KUKA KRL program: f1_Kuka_APT220T03S20.SRC

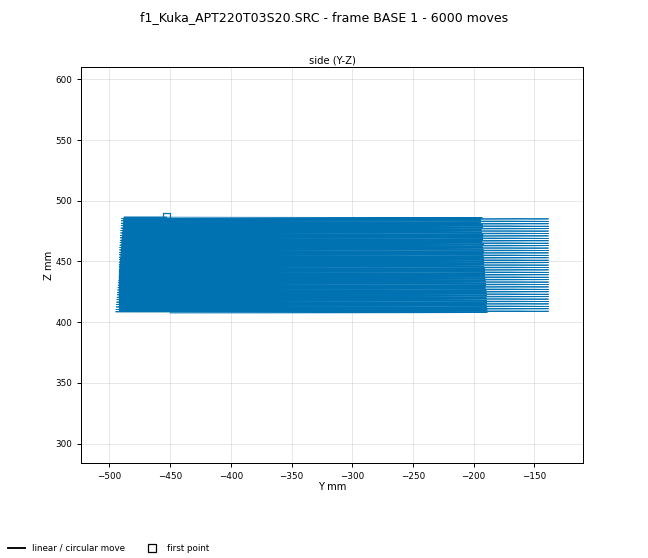
[picture p0: tool path of f1_Kuka_APT220T03S20.SRC in frame BASE 1, 6000 of 6001 moves have a stored position in this frame; points joined in program order, loops and branches not executed]
&ACCESS RVP
&REL 2
&PARAM TEMPLATE = C:\KRC\Roboter\Template\vorgabe
&PARAM EDITMASK = *
DEF f1_Kuka_APT220T03S20()


;FOLD INI;%{PE}%V3.2.0,%MKUKATPBASIS,%CINIT,%VCOMMON,%P
  ;FOLD BAS INI;%{E}%V3.2.0,%MKUKATPBASIS,%CINIT,%VINIT,%P
    GLOBAL INTERRUPT DECL 3 WHEN $STOPMESS==TRUE DO IR_STOPM ( )
    INTERRUPT ON 3
    BAS (#INITMOV,0 )
  ;ENDFOLD (BAS INI)
  ;FOLD USER INI;%{E}%V3.2.0,%MKUKATPUSER,%CINIT,%VINIT,%P
    ;Make your modifications here
  ;ENDFOLD (USER INI)
;ENDFOLD (INI)


;*** Make Null PTP Move
  PTP $pos_act

;*** Auto Load The Correct TOOL Data
  $tool=tool_data[3]

;*** Auto Load The Correct BASE Data
  $base=base_data[1]

  $ADVANCE = 5

;*** Restate Last Velocity
MMPM(30000.0)
SetRPM(6000)
LIN {X -0.066,Y -453.001,Z 486.562,A 0.000,B 0.000,C 90.000,E1 101.130} C_DIS
LIN {X -0.099,Y -473.711,Z 486.551,A 0.000,B 0.000,C 90.000,E1 99.265} C_DIS
LIN {X 0.194,Y -481.469,Z 486.548,A 0.000,B 0.000,C 90.000,E1 98.568} C_DIS
LIN {X 0.203,Y -483.436,Z 486.546,A 0.000,B 0.000,C 90.000,E1 98.341} C_DIS
LIN {X -0.197,Y -484.945,Z 486.545,A 0.000,B 0.000,C 90.000,E1 98.163} C_DIS
LIN {X 0.167,Y -486.209,Z 486.544,A 0.000,B 0.000,C 90.000,E1 97.871} C_DIS
LIN {X -0.015,Y -487.138,Z 486.542,A 0.000,B 0.000,C 90.000,E1 97.644} C_DIS
LIN {X 0.186,Y -488.149,Z 486.540,A 0.000,B 0.000,C 90.000,E1 97.125} C_DIS
LIN {X -0.091,Y -488.162,Z 486.537,A 0.000,B 0.000,C 90.000,E1 96.663} C_DIS
LIN {X 0.122,Y -487.175,Z 486.534,A 0.000,B 0.000,C 90.000,E1 96.144} C_DIS
LIN {X 0.010,Y -486.265,Z 486.533,A 0.000,B 0.000,C 90.000,E1 95.910} C_DIS
LIN {X -0.151,Y -485.019,Z 486.531,A 0.000,B 0.000,C 90.000,E1 95.682} C_DIS
LIN {X 0.212,Y -483.351,Z 486.530,A 0.000,B 0.000,C 90.000,E1 95.391} C_DIS
LIN {X 0.076,Y -465.274,Z 486.518,A 0.000,B 0.000,C 90.000,E1 93.154} C_DIS
LIN {X 0.213,Y -454.119,Z 486.509,A 0.000,B 0.000,C 90.000,E1 91.604} C_DIS
LIN {X 0.144,Y -435.760,Z 486.493,A 0.000,B 0.000,C 90.000,E1 88.740} C_DIS
LIN {X 0.163,Y -421.080,Z 486.480,A 0.000,B 0.000,C 90.000,E1 86.331} C_DIS
LIN {X 0.167,Y -408.275,Z 486.468,A 0.000,B 0.000,C 90.000,E1 84.147} C_DIS
LIN {X -0.037,Y -395.778,Z 486.455,A 0.000,B 0.000,C 90.000,E1 81.951} C_DIS
LIN {X -0.125,Y -384.823,Z 486.444,A 0.000,B 0.000,C 90.000,E1 79.982} C_DIS
LIN {X 0.074,Y -369.281,Z 486.428,A 0.000,B 0.000,C 90.000,E1 77.061} C_DIS
LIN {X 0.055,Y -357.557,Z 486.415,A 0.000,B 0.000,C 90.000,E1 74.700} C_DIS
LIN {X -0.046,Y -347.157,Z 486.402,A 0.000,B 0.000,C 90.000,E1 72.308} C_DIS
LIN {X 0.119,Y -333.448,Z 486.381,A 0.000,B 0.000,C 90.000,E1 68.592} C_DIS
LIN {X 0.012,Y -323.935,Z 486.366,A 0.000,B 0.000,C 90.000,E1 65.793} C_DIS
LIN {X -0.012,Y -315.733,Z 486.351,A 0.000,B 0.000,C 90.000,E1 63.256} C_DIS
LIN {X 0.042,Y -307.567,Z 486.337,A 0.000,B 0.000,C 90.000,E1 60.667} C_DIS
LIN {X 0.124,Y -297.594,Z 486.319,A 0.000,B 0.000,C 90.000,E1 57.375} C_DIS
LIN {X -0.027,Y -288.131,Z 486.300,A 0.000,B 0.000,C 90.000,E1 54.069} C_DIS
LIN {X 0.029,Y -282.669,Z 486.289,A 0.000,B 0.000,C 90.000,E1 52.029} C_DIS
LIN {X -0.014,Y -277.048,Z 486.278,A 0.000,B 0.000,C 90.000,E1 49.989} C_DIS
LIN {X -0.019,Y -270.999,Z 486.266,A 0.000,B 0.000,C 90.000,E1 47.919} C_DIS
LIN {X 0.045,Y -264.538,Z 486.255,A 0.000,B 0.000,C 90.000,E1 45.810} C_DIS
LIN {X -0.028,Y -257.779,Z 486.243,A 0.000,B 0.000,C 90.000,E1 43.704} C_DIS
LIN {X -0.024,Y -248.806,Z 486.227,A 0.000,B 0.000,C 90.000,E1 40.825} C_DIS
LIN {X 0.021,Y -240.234,Z 486.211,A 0.000,B 0.000,C 90.000,E1 37.890} C_DIS
LIN {X 0.095,Y -232.095,Z 486.194,A 0.000,B 0.000,C 90.000,E1 34.898} C_DIS
LIN {X 0.084,Y -224.777,Z 486.177,A 0.000,B 0.000,C 90.000,E1 31.878} C_DIS
LIN {X 0.039,Y -218.459,Z 486.160,A 0.000,B 0.000,C 90.000,E1 28.821} C_DIS
LIN {X 0.011,Y -212.877,Z 486.143,A 0.000,B 0.000,C 90.000,E1 25.720} C_DIS
LIN {X 0.061,Y -207.080,Z 486.121,A 0.000,B 0.000,C 90.000,E1 21.770} C_DIS
LIN {X -0.059,Y -202.295,Z 486.099,A 0.000,B 0.000,C 90.000,E1 17.819} C_DIS
LIN {X 0.019,Y -198.439,Z 486.077,A 0.000,B 0.000,C 90.000,E1 13.772} C_DIS
LIN {X -0.032,Y -195.236,Z 486.049,A 0.000,B 0.000,C 90.000,E1 8.916} C_DIS
LIN {X -0.003,Y -192.924,Z 486.009,A 0.000,B 0.000,C 90.000,E1 1.547} C_DIS
LIN {X 0.083,Y -194.698,Z 485.956,A 0.000,B 0.000,C 90.000,E1 352.129} C_DIS
LIN {X 0.104,Y -197.850,Z 485.929,A 0.000,B 0.000,C 90.000,E1 347.229} C_DIS
LIN {X -0.053,Y -202.300,Z 485.902,A 0.000,B 0.000,C 90.000,E1 342.417} C_DIS
LIN {X -0.067,Y -207.060,Z 485.880,A 0.000,B 0.000,C 90.000,E1 338.411} C_DIS
LIN {X 0.066,Y -212.566,Z 485.858,A 0.000,B 0.000,C 90.000,E1 334.409} C_DIS
LIN {X -0.012,Y -218.738,Z 485.836,A 0.000,B 0.000,C 90.000,E1 330.511} C_DIS
LIN {X 0.052,Y -225.483,Z 485.815,A 0.000,B 0.000,C 90.000,E1 326.628} C_DIS
LIN {X -0.056,Y -232.921,Z 485.793,A 0.000,B 0.000,C 90.000,E1 322.844} C_DIS
LIN {X -0.070,Y -241.150,Z 485.773,A 0.000,B 0.000,C 90.000,E1 319.094} C_DIS
LIN {X -0.057,Y -248.484,Z 485.756,A 0.000,B 0.000,C 90.000,E1 316.134} C_DIS
LIN {X 0.002,Y -257.837,Z 485.738,A 0.000,B 0.000,C 90.000,E1 312.852} C_DIS
LIN {X 0.080,Y -269.299,Z 485.718,A 0.000,B 0.000,C 90.000,E1 309.277} C_DIS
LIN {X 0.060,Y -282.037,Z 485.699,A 0.000,B 0.000,C 90.000,E1 305.804} C_DIS
LIN {X 0.021,Y -295.837,Z 485.680,A 0.000,B 0.000,C 90.000,E1 302.418} C_DIS
LIN {X -0.105,Y -309.070,Z 485.664,A 0.000,B 0.000,C 90.000,E1 299.461} C_DIS
LIN {X -0.041,Y -320.167,Z 485.651,A 0.000,B 0.000,C 90.000,E1 297.180} C_DIS
LIN {X -0.087,Y -336.107,Z 485.635,A 0.000,B 0.000,C 90.000,E1 294.335} C_DIS
LIN {X 0.044,Y -351.864,Z 485.621,A 0.000,B 0.000,C 90.000,E1 291.844} C_DIS
LIN {X -0.013,Y -369.266,Z 485.608,A 0.000,B 0.000,C 90.000,E1 289.450} C_DIS
LIN {X 0.122,Y -388.273,Z 485.595,A 0.000,B 0.000,C 90.000,E1 287.094} C_DIS
LIN {X -0.021,Y -410.726,Z 485.581,A 0.000,B 0.000,C 90.000,E1 284.592} C_DIS
LIN {X -0.224,Y -426.019,Z 485.572,A 0.000,B 0.000,C 90.000,E1 283.008} C_DIS
LIN {X -0.004,Y -438.423,Z 485.565,A 0.000,B 0.000,C 90.000,E1 281.658} C_DIS
LIN {X -0.012,Y -448.140,Z 485.559,A 0.000,B 0.000,C 90.000,E1 280.602} C_DIS
LIN {X 0.192,Y -454.892,Z 485.555,A 0.000,B 0.000,C 90.000,E1 279.792} C_DIS
LIN {X 0.079,Y -461.053,Z 485.550,A 0.000,B 0.000,C 90.000,E1 279.029} C_DIS
LIN {X -0.054,Y -466.674,Z 485.546,A 0.000,B 0.000,C 90.000,E1 278.276} C_DIS
LIN {X -0.208,Y -471.720,Z 485.542,A 0.000,B 0.000,C 90.000,E1 277.530} C_DIS
LIN {X 0.223,Y -476.192,Z 485.537,A 0.000,B 0.000,C 90.000,E1 276.720} C_DIS
LIN {X 0.215,Y -480.149,Z 485.533,A 0.000,B 0.000,C 90.000,E1 275.967} C_DIS
LIN {X -0.156,Y -482.500,Z 485.531,A 0.000,B 0.000,C 90.000,E1 275.511} C_DIS
LIN {X 0.016,Y -484.512,Z 485.528,A 0.000,B 0.000,C 90.000,E1 274.992} C_DIS
LIN {X 0.193,Y -486.239,Z 485.525,A 0.000,B 0.000,C 90.000,E1 274.473} C_DIS
LIN {X -0.105,Y -487.676,Z 485.522,A 0.000,B 0.000,C 90.000,E1 274.012} C_DIS
LIN {X 0.058,Y -488.770,Z 485.519,A 0.000,B 0.000,C 90.000,E1 273.498} C_DIS
LIN {X -0.227,Y -489.533,Z 485.517,A 0.000,B 0.000,C 90.000,E1 273.037} C_DIS
LIN {X -0.044,Y -489.993,Z 485.514,A 0.000,B 0.000,C 90.000,E1 272.522} C_DIS
LIN {X 0.146,Y -490.072,Z 485.511,A 0.000,B 0.000,C 90.000,E1 272.007} C_DIS
LIN {X -0.134,Y -489.708,Z 485.509,A 0.000,B 0.000,C 90.000,E1 271.547} C_DIS
LIN {X 0.060,Y -488.939,Z 485.506,A 0.000,B 0.000,C 90.000,E1 271.031} C_DIS
LIN {X -0.235,Y -487.615,Z 485.503,A 0.000,B 0.000,C 90.000,E1 270.573} C_DIS
LIN {X -0.046,Y -485.714,Z 485.500,A 0.000,B 0.000,C 90.000,E1 270.057} C_DIS
LIN {X 0.134,Y -483.153,Z 485.498,A 0.000,B 0.000,C 90.000,E1 269.542} C_DIS
LIN {X -0.186,Y -479.844,Z 485.495,A 0.000,B 0.000,C 90.000,E1 269.083} C_DIS
LIN {X -0.043,Y -475.615,Z 485.492,A 0.000,B 0.000,C 90.000,E1 268.568} C_DIS
LIN {X 0.091,Y -470.396,Z 485.489,A 0.000,B 0.000,C 90.000,E1 268.051} C_DIS
LIN {X 0.002,Y -464.305,Z 485.487,A 0.000,B 0.000,C 90.000,E1 267.593} C_DIS
LIN {X -0.231,Y -461.262,Z 485.486,A 0.000,B 0.000,C 90.000,E1 267.421} C_DIS
LIN {X 0.033,Y -454.595,Z 485.483,A 0.000,B 0.000,C 90.000,E1 267.020} C_DIS
LIN {X -0.113,Y -447.751,Z 485.482,A 0.000,B 0.000,C 90.000,E1 266.731} C_DIS
LIN {X 0.088,Y -440.644,Z 485.480,A 0.000,B 0.000,C 90.000,E1 266.445} C_DIS
LIN {X -0.218,Y -432.837,Z 485.479,A 0.000,B 0.000,C 90.000,E1 266.274} C_DIS
LIN {X -0.101,Y -424.190,Z 485.478,A 0.000,B 0.000,C 90.000,E1 266.102} C_DIS
LIN {X -0.056,Y -413.858,Z 485.478,A 0.000,B 0.000,C 90.000,E1 265.988} C_DIS
LIN {X -0.214,Y -409.409,Z 485.478,A 0.000,B 0.000,C 90.000,E1 265.988} C_DIS
LIN {X 0.063,Y -180.918,Z 485.477,A 0.000,B 0.000,C 90.000,E1 265.927} C_DIS
LIN {X -0.088,Y -180.843,Z 485.472,A 0.000,B 0.000,C 90.000,E1 264.951} C_DIS
LIN {X -0.011,Y -178.885,Z 485.443,A 0.000,B 0.000,C 90.000,E1 259.690} C_DIS
LIN {X 0.064,Y -175.928,Z 485.414,A 0.000,B 0.000,C 90.000,E1 254.574} C_DIS
LIN {X 0.009,Y -175.370,Z 485.410,A 0.000,B 0.000,C 90.000,E1 253.740} C_DIS
LIN {X 0.067,Y -172.147,Z 485.386,A 0.000,B 0.000,C 90.000,E1 249.444} C_DIS
LIN {X 0.045,Y -171.612,Z 485.381,A 0.000,B 0.000,C 90.000,E1 248.592} C_DIS
LIN {X 0.033,Y -167.834,Z 485.357,A 0.000,B 0.000,C 90.000,E1 244.280} C_DIS
LIN {X 0.050,Y -166.561,Z 485.348,A 0.000,B 0.000,C 90.000,E1 242.538} C_DIS
LIN {X -0.040,Y -162.555,Z 485.323,A 0.000,B 0.000,C 90.000,E1 238.201} C_DIS
LIN {X 0.020,Y -161.234,Z 485.313,A 0.000,B 0.000,C 90.000,E1 236.421} C_DIS
LIN {X 0.054,Y -157.239,Z 485.289,A 0.000,B 0.000,C 90.000,E1 231.984} C_DIS
LIN {X -0.022,Y -155.962,Z 485.279,A 0.000,B 0.000,C 90.000,E1 230.231} C_DIS
LIN {X 0.036,Y -152.217,Z 485.254,A 0.000,B 0.000,C 90.000,E1 225.729} C_DIS
LIN {X 0.056,Y -150.461,Z 485.239,A 0.000,B 0.000,C 90.000,E1 223.014} C_DIS
LIN {X 0.082,Y -147.186,Z 485.214,A 0.000,B 0.000,C 90.000,E1 218.463} C_DIS
LIN {X 0.049,Y -145.204,Z 485.194,A 0.000,B 0.000,C 90.000,E1 214.818} C_DIS
LIN {X -0.041,Y -142.340,Z 485.163,A 0.000,B 0.000,C 90.000,E1 209.333} C_DIS
LIN {X 0.012,Y -141.728,Z 485.153,A 0.000,B 0.000,C 90.000,E1 207.462} C_DIS
LIN {X -0.006,Y -139.482,Z 485.116,A 0.000,B 0.000,C 90.000,E1 200.972} C_DIS
LIN {X -0.017,Y -138.980,Z 485.101,A 0.000,B 0.000,C 90.000,E1 198.181} C_DIS
LIN {X -0.056,Y -138.333,Z 485.054,A 0.000,B 0.000,C 90.000,E1 189.792} C_DIS
LIN {X -0.032,Y -139.428,Z 485.008,A 0.000,B 0.000,C 90.000,E1 181.375} C_DIS
LIN {X 0.022,Y -141.355,Z 484.971,A 0.000,B 0.000,C 90.000,E1 174.837} C_DIS
LIN {X -0.002,Y -142.708,Z 484.956,A 0.000,B 0.000,C 90.000,E1 172.064} C_DIS
LIN {X -0.043,Y -145.082,Z 484.930,A 0.000,B 0.000,C 90.000,E1 167.465} C_DIS
LIN {X -0.047,Y -147.707,Z 484.910,A 0.000,B 0.000,C 90.000,E1 163.795} C_DIS
LIN {X 0.036,Y -150.361,Z 484.890,A 0.000,B 0.000,C 90.000,E1 160.115} C_DIS
LIN {X 0.054,Y -153.786,Z 484.869,A 0.000,B 0.000,C 90.000,E1 156.485} C_DIS
LIN {X -0.025,Y -157.198,Z 484.850,A 0.000,B 0.000,C 90.000,E1 152.922} C_DIS
LIN {X 0.057,Y -161.360,Z 484.830,A 0.000,B 0.000,C 90.000,E1 149.331} C_DIS
LIN {X 0.068,Y -165.562,Z 484.810,A 0.000,B 0.000,C 90.000,E1 145.801} C_DIS
LIN {X -0.048,Y -170.478,Z 484.791,A 0.000,B 0.000,C 90.000,E1 142.351} C_DIS
LIN {X 0.101,Y -175.360,Z 484.772,A 0.000,B 0.000,C 90.000,E1 138.852} C_DIS
LIN {X -0.035,Y -180.985,Z 484.753,A 0.000,B 0.000,C 90.000,E1 135.486} C_DIS
LIN {X -0.049,Y -186.409,Z 484.734,A 0.000,B 0.000,C 90.000,E1 132.123} C_DIS
LIN {X -0.110,Y -191.038,Z 484.720,A 0.000,B 0.000,C 90.000,E1 129.644} C_DIS
LIN {X 0.023,Y -193.423,Z 484.712,A 0.000,B 0.000,C 90.000,E1 128.177} C_DIS
LIN {X -0.005,Y -291.168,Z 484.712,A 0.000,B 0.000,C 90.000,E1 128.177} C_DIS
LIN {X -0.085,Y -292.124,Z 484.712,A 0.000,B 0.000,C 90.000,E1 128.177} C_DIS
LIN {X -0.050,Y -296.671,Z 484.711,A 0.000,B 0.000,C 90.000,E1 127.971} C_DIS
LIN {X 0.020,Y -299.838,Z 484.709,A 0.000,B 0.000,C 90.000,E1 127.684} C_DIS
LIN {X 0.147,Y -303.532,Z 484.707,A 0.000,B 0.000,C 90.000,E1 127.156} C_DIS
LIN {X -0.090,Y -305.238,Z 484.705,A 0.000,B 0.000,C 90.000,E1 126.870} C_DIS
LIN {X 0.101,Y -306.580,Z 484.703,A 0.000,B 0.000,C 90.000,E1 126.503} C_DIS
LIN {X -0.077,Y -317.797,Z 484.683,A 0.000,B 0.000,C 90.000,E1 122.959} C_DIS
LIN {X -0.030,Y -328.281,Z 484.667,A 0.000,B 0.000,C 90.000,E1 120.079} C_DIS
LIN {X -0.002,Y -340.128,Z 484.651,A 0.000,B 0.000,C 90.000,E1 117.257} C_DIS
LIN {X -0.116,Y -353.449,Z 484.636,A 0.000,B 0.000,C 90.000,E1 114.515} C_DIS
LIN {X 0.108,Y -366.623,Z 484.623,A 0.000,B 0.000,C 90.000,E1 112.078} C_DIS
LIN {X -0.082,Y -381.150,Z 484.610,A 0.000,B 0.000,C 90.000,E1 109.758} C_DIS
LIN {X -0.040,Y -397.136,Z 484.597,A 0.000,B 0.000,C 90.000,E1 107.457} C_DIS
LIN {X 0.171,Y -414.700,Z 484.585,A 0.000,B 0.000,C 90.000,E1 105.190} C_DIS
LIN {X -0.185,Y -433.943,Z 484.572,A 0.000,B 0.000,C 90.000,E1 103.063} C_DIS
LIN {X 0.027,Y -454.145,Z 484.561,A 0.000,B 0.000,C 90.000,E1 101.007} C_DIS
LIN {X -0.012,Y -474.885,Z 484.551,A 0.000,B 0.000,C 90.000,E1 99.151} C_DIS
LIN {X 0.167,Y -480.145,Z 484.548,A 0.000,B 0.000,C 90.000,E1 98.690} C_DIS
LIN {X -0.145,Y -482.402,Z 484.547,A 0.000,B 0.000,C 90.000,E1 98.511} C_DIS
LIN {X 0.018,Y -484.116,Z 484.546,A 0.000,B 0.000,C 90.000,E1 98.276} C_DIS
LIN {X -0.170,Y -485.628,Z 484.545,A 0.000,B 0.000,C 90.000,E1 98.049} C_DIS
LIN {X 0.193,Y -486.758,Z 484.543,A 0.000,B 0.000,C 90.000,E1 97.757} C_DIS
LIN {X -0.095,Y -488.102,Z 484.540,A 0.000,B 0.000,C 90.000,E1 97.296} C_DIS
LIN {X 0.109,Y -488.413,Z 484.538,A 0.000,B 0.000,C 90.000,E1 96.777} C_DIS
LIN {X -0.164,Y -487.742,Z 484.535,A 0.000,B 0.000,C 90.000,E1 96.315} C_DIS
LIN {X 0.049,Y -485.978,Z 484.532,A 0.000,B 0.000,C 90.000,E1 95.796} C_DIS
LIN {X -0.112,Y -484.583,Z 484.531,A 0.000,B 0.000,C 90.000,E1 95.568} C_DIS
LIN {X -0.079,Y -478.706,Z 484.527,A 0.000,B 0.000,C 90.000,E1 94.821} C_DIS
LIN {X 0.175,Y -460.878,Z 484.514,A 0.000,B 0.000,C 90.000,E1 92.522} C_DIS
LIN {X -0.020,Y -448.423,Z 484.504,A 0.000,B 0.000,C 90.000,E1 90.745} C_DIS
LIN {X 0.149,Y -435.261,Z 484.492,A 0.000,B 0.000,C 90.000,E1 88.625} C_DIS
LIN {X 0.149,Y -420.581,Z 484.479,A 0.000,B 0.000,C 90.000,E1 86.216} C_DIS
LIN {X -0.158,Y -406.238,Z 484.465,A 0.000,B 0.000,C 90.000,E1 83.799} C_DIS
LIN {X -0.078,Y -395.315,Z 484.455,A 0.000,B 0.000,C 90.000,E1 81.837} C_DIS
LIN {X -0.108,Y -384.376,Z 484.444,A 0.000,B 0.000,C 90.000,E1 79.859} C_DIS
LIN {X 0.088,Y -368.860,Z 484.427,A 0.000,B 0.000,C 90.000,E1 76.937} C_DIS
LIN {X 0.066,Y -357.181,Z 484.414,A 0.000,B 0.000,C 90.000,E1 74.574} C_DIS
LIN {X -0.038,Y -346.833,Z 484.401,A 0.000,B 0.000,C 90.000,E1 72.181} C_DIS
LIN {X 0.131,Y -334.216,Z 484.382,A 0.000,B 0.000,C 90.000,E1 68.773} C_DIS
LIN {X -0.036,Y -322.537,Z 484.363,A 0.000,B 0.000,C 90.000,E1 65.357} C_DIS
LIN {X 0.044,Y -316.364,Z 484.352,A 0.000,B 0.000,C 90.000,E1 63.435} C_DIS
LIN {X 0.118,Y -308.153,Z 484.338,A 0.000,B 0.000,C 90.000,E1 60.845} C_DIS
LIN {X 0.068,Y -298.121,Z 484.320,A 0.000,B 0.000,C 90.000,E1 57.582} C_DIS
LIN {X -0.065,Y -288.589,Z 484.301,A 0.000,B 0.000,C 90.000,E1 54.276} C_DIS
LIN {X -0.172,Y -283.117,Z 484.290,A 0.000,B 0.000,C 90.000,E1 52.271} C_DIS
LIN {X -0.029,Y -277.516,Z 484.279,A 0.000,B 0.000,C 90.000,E1 50.194} C_DIS
LIN {X 0.000,Y -271.503,Z 484.267,A 0.000,B 0.000,C 90.000,E1 48.119} C_DIS
LIN {X -0.126,Y -265.082,Z 484.256,A 0.000,B 0.000,C 90.000,E1 46.053} C_DIS
LIN {X 0.003,Y -258.374,Z 484.244,A 0.000,B 0.000,C 90.000,E1 43.905} C_DIS
LIN {X 0.018,Y -248.304,Z 484.226,A 0.000,B 0.000,C 90.000,E1 40.663} C_DIS
LIN {X 0.027,Y -238.693,Z 484.208,A 0.000,B 0.000,C 90.000,E1 37.363} C_DIS
LIN {X -0.075,Y -230.694,Z 484.191,A 0.000,B 0.000,C 90.000,E1 34.405} C_DIS
LIN {X 0.071,Y -223.578,Z 484.174,A 0.000,B 0.000,C 90.000,E1 31.337} C_DIS
LIN {X -0.007,Y -217.384,Z 484.157,A 0.000,B 0.000,C 90.000,E1 28.281} C_DIS
LIN {X 0.032,Y -211.971,Z 484.140,A 0.000,B 0.000,C 90.000,E1 25.155} C_DIS
LIN {X -0.023,Y -206.290,Z 484.118,A 0.000,B 0.000,C 90.000,E1 21.227} C_DIS
LIN {X 0.032,Y -201.634,Z 484.096,A 0.000,B 0.000,C 90.000,E1 17.221} C_DIS
LIN {X 0.086,Y -197.927,Z 484.073,A 0.000,B 0.000,C 90.000,E1 13.175} C_DIS
LIN {X -0.077,Y -194.481,Z 484.042,A 0.000,B 0.000,C 90.000,E1 7.530} C_DIS
LIN {X 0.057,Y -195.445,Z 483.947,A 0.000,B 0.000,C 90.000,E1 350.500} C_DIS
LIN {X -0.044,Y -199.071,Z 483.920,A 0.000,B 0.000,C 90.000,E1 345.644} C_DIS
LIN {X 0.033,Y -203.010,Z 483.898,A 0.000,B 0.000,C 90.000,E1 341.583} C_DIS
LIN {X -0.007,Y -207.968,Z 483.875,A 0.000,B 0.000,C 90.000,E1 337.592} C_DIS
LIN {X -0.031,Y -213.585,Z 483.854,A 0.000,B 0.000,C 90.000,E1 333.640} C_DIS
LIN {X -0.084,Y -219.884,Z 483.832,A 0.000,B 0.000,C 90.000,E1 329.744} C_DIS
LIN {X -0.064,Y -226.774,Z 483.810,A 0.000,B 0.000,C 90.000,E1 325.881} C_DIS
LIN {X -0.005,Y -234.402,Z 483.789,A 0.000,B 0.000,C 90.000,E1 322.065} C_DIS
LIN {X -0.003,Y -242.796,Z 483.768,A 0.000,B 0.000,C 90.000,E1 318.324} C_DIS
LIN {X 0.052,Y -251.380,Z 483.750,A 0.000,B 0.000,C 90.000,E1 315.000} C_DIS
LIN {X 0.027,Y -261.066,Z 483.732,A 0.000,B 0.000,C 90.000,E1 311.757} C_DIS
LIN {X -0.046,Y -271.684,Z 483.714,A 0.000,B 0.000,C 90.000,E1 308.588} C_DIS
LIN {X 0.061,Y -284.676,Z 483.695,A 0.000,B 0.000,C 90.000,E1 305.105} C_DIS
LIN {X -0.053,Y -298.724,Z 483.676,A 0.000,B 0.000,C 90.000,E1 301.750} C_DIS
LIN {X 0.073,Y -313.690,Z 483.658,A 0.000,B 0.000,C 90.000,E1 298.437} C_DIS
LIN {X 0.169,Y -323.588,Z 483.647,A 0.000,B 0.000,C 90.000,E1 296.488} C_DIS
LIN {X -0.070,Y -339.930,Z 483.632,A 0.000,B 0.000,C 90.000,E1 293.695} C_DIS
LIN {X -0.008,Y -353.980,Z 483.620,A 0.000,B 0.000,C 90.000,E1 291.535} C_DIS
LIN {X -0.099,Y -369.308,Z 483.608,A 0.000,B 0.000,C 90.000,E1 289.450} C_DIS
LIN {X 0.033,Y -388.293,Z 483.595,A 0.000,B 0.000,C 90.000,E1 287.094} C_DIS
LIN {X -0.109,Y -410.777,Z 483.581,A 0.000,B 0.000,C 90.000,E1 284.592} C_DIS
LIN {X -0.177,Y -425.949,Z 483.572,A 0.000,B 0.000,C 90.000,E1 283.008} C_DIS
LIN {X 0.129,Y -438.298,Z 483.565,A 0.000,B 0.000,C 90.000,E1 281.658} C_DIS
LIN {X -0.049,Y -445.608,Z 483.560,A 0.000,B 0.000,C 90.000,E1 280.894} C_DIS
LIN {X 0.157,Y -452.543,Z 483.556,A 0.000,B 0.000,C 90.000,E1 280.084} C_DIS
LIN {X 0.032,Y -458.939,Z 483.552,A 0.000,B 0.000,C 90.000,E1 279.321} C_DIS
LIN {X 0.168,Y -466.548,Z 483.546,A 0.000,B 0.000,C 90.000,E1 278.276} C_DIS
LIN {X 0.015,Y -471.623,Z 483.542,A 0.000,B 0.000,C 90.000,E1 277.530} C_DIS
LIN {X -0.026,Y -476.156,Z 483.538,A 0.000,B 0.000,C 90.000,E1 276.777} C_DIS
LIN {X -0.088,Y -480.145,Z 483.533,A 0.000,B 0.000,C 90.000,E1 276.030} C_DIS
LIN {X 0.070,Y -482.488,Z 483.531,A 0.000,B 0.000,C 90.000,E1 275.511} C_DIS
LIN {X -0.241,Y -484.529,Z 483.528,A 0.000,B 0.000,C 90.000,E1 275.049} C_DIS
LIN {X -0.064,Y -486.287,Z 483.525,A 0.000,B 0.000,C 90.000,E1 274.531} C_DIS
LIN {X 0.123,Y -487.727,Z 483.522,A 0.000,B 0.000,C 90.000,E1 274.012} C_DIS
LIN {X -0.201,Y -488.884,Z 483.520,A 0.000,B 0.000,C 90.000,E1 273.555} C_DIS
LIN {X 0.002,Y -489.645,Z 483.517,A 0.000,B 0.000,C 90.000,E1 273.037} C_DIS
LIN {X 0.186,Y -490.105,Z 483.514,A 0.000,B 0.000,C 90.000,E1 272.522} C_DIS
LIN {X -0.113,Y -490.201,Z 483.511,A 0.000,B 0.000,C 90.000,E1 272.064} C_DIS
LIN {X 0.098,Y -489.875,Z 483.509,A 0.000,B 0.000,C 90.000,E1 271.547} C_DIS
LIN {X -0.197,Y -489.145,Z 483.506,A 0.000,B 0.000,C 90.000,E1 271.088} C_DIS
LIN {X -0.003,Y -487.837,Z 483.503,A 0.000,B 0.000,C 90.000,E1 270.573} C_DIS
LIN {X 0.187,Y -485.979,Z 483.500,A 0.000,B 0.000,C 90.000,E1 270.057} C_DIS
LIN {X -0.116,Y -483.442,Z 483.498,A 0.000,B 0.000,C 90.000,E1 269.599} C_DIS
LIN {X 0.047,Y -480.160,Z 483.495,A 0.000,B 0.000,C 90.000,E1 269.083} C_DIS
LIN {X -0.120,Y -478.231,Z 483.494,A 0.000,B 0.000,C 90.000,E1 268.854} C_DIS
LIN {X 0.013,Y -473.551,Z 483.491,A 0.000,B 0.000,C 90.000,E1 268.339} C_DIS
LIN {X -0.187,Y -468.011,Z 483.488,A 0.000,B 0.000,C 90.000,E1 267.879} C_DIS
LIN {X -0.007,Y -461.773,Z 483.486,A 0.000,B 0.000,C 90.000,E1 267.421} C_DIS
LIN {X 0.218,Y -455.153,Z 483.484,A 0.000,B 0.000,C 90.000,E1 267.020} C_DIS
LIN {X 0.020,Y -448.307,Z 483.482,A 0.000,B 0.000,C 90.000,E1 266.731} C_DIS
LIN {X 0.175,Y -441.166,Z 483.480,A 0.000,B 0.000,C 90.000,E1 266.445} C_DIS
LIN {X -0.151,Y -433.386,Z 483.479,A 0.000,B 0.000,C 90.000,E1 266.274} C_DIS
LIN {X -0.038,Y -425.010,Z 483.478,A 0.000,B 0.000,C 90.000,E1 266.102} C_DIS
LIN {X 0.004,Y -415.303,Z 483.478,A 0.000,B 0.000,C 90.000,E1 265.988} C_DIS
LIN {X 0.175,Y -409.435,Z 483.478,A 0.000,B 0.000,C 90.000,E1 265.931} C_DIS
LIN {X 0.055,Y -180.918,Z 483.477,A 0.000,B 0.000,C 90.000,E1 265.927} C_DIS
LIN {X 0.085,Y -180.842,Z 483.472,A 0.000,B 0.000,C 90.000,E1 264.894} C_DIS
LIN {X -0.019,Y -178.885,Z 483.443,A 0.000,B 0.000,C 90.000,E1 259.690} C_DIS
LIN {X 0.058,Y -175.927,Z 483.414,A 0.000,B 0.000,C 90.000,E1 254.574} C_DIS
LIN {X 0.003,Y -175.368,Z 483.410,A 0.000,B 0.000,C 90.000,E1 253.740} C_DIS
LIN {X 0.061,Y -172.145,Z 483.386,A 0.000,B 0.000,C 90.000,E1 249.444} C_DIS
LIN {X 0.039,Y -171.610,Z 483.381,A 0.000,B 0.000,C 90.000,E1 248.592} C_DIS
LIN {X 0.026,Y -167.833,Z 483.357,A 0.000,B 0.000,C 90.000,E1 244.280} C_DIS
LIN {X 0.044,Y -166.559,Z 483.348,A 0.000,B 0.000,C 90.000,E1 242.538} C_DIS
LIN {X -0.046,Y -162.553,Z 483.323,A 0.000,B 0.000,C 90.000,E1 238.201} C_DIS
LIN {X 0.014,Y -161.232,Z 483.313,A 0.000,B 0.000,C 90.000,E1 236.421} C_DIS
LIN {X 0.049,Y -157.237,Z 483.289,A 0.000,B 0.000,C 90.000,E1 231.984} C_DIS
LIN {X -0.028,Y -155.962,Z 483.279,A 0.000,B 0.000,C 90.000,E1 230.231} C_DIS
LIN {X 0.030,Y -152.215,Z 483.254,A 0.000,B 0.000,C 90.000,E1 225.729} C_DIS
LIN {X 0.051,Y -150.460,Z 483.239,A 0.000,B 0.000,C 90.000,E1 223.014} C_DIS
LIN {X 0.077,Y -147.184,Z 483.214,A 0.000,B 0.000,C 90.000,E1 218.463} C_DIS
LIN {X 0.043,Y -145.203,Z 483.194,A 0.000,B 0.000,C 90.000,E1 214.818} C_DIS
LIN {X -0.047,Y -142.339,Z 483.163,A 0.000,B 0.000,C 90.000,E1 209.333} C_DIS
LIN {X 0.006,Y -141.727,Z 483.153,A 0.000,B 0.000,C 90.000,E1 207.462} C_DIS
LIN {X -0.012,Y -139.480,Z 483.116,A 0.000,B 0.000,C 90.000,E1 200.972} C_DIS
LIN {X -0.022,Y -138.980,Z 483.101,A 0.000,B 0.000,C 90.000,E1 198.181} C_DIS
LIN {X -0.038,Y -138.332,Z 483.054,A 0.000,B 0.000,C 90.000,E1 189.782} C_DIS
LIN {X -0.037,Y -139.428,Z 483.008,A 0.000,B 0.000,C 90.000,E1 181.375} C_DIS
LIN {X 0.016,Y -141.355,Z 482.971,A 0.000,B 0.000,C 90.000,E1 174.837} C_DIS
LIN {X -0.008,Y -142.709,Z 482.956,A 0.000,B 0.000,C 90.000,E1 172.064} C_DIS
LIN {X -0.049,Y -145.083,Z 482.930,A 0.000,B 0.000,C 90.000,E1 167.465} C_DIS
LIN {X -0.053,Y -147.708,Z 482.910,A 0.000,B 0.000,C 90.000,E1 163.795} C_DIS
LIN {X 0.031,Y -150.363,Z 482.890,A 0.000,B 0.000,C 90.000,E1 160.115} C_DIS
LIN {X 0.049,Y -153.788,Z 482.869,A 0.000,B 0.000,C 90.000,E1 156.485} C_DIS
LIN {X -0.031,Y -157.201,Z 482.850,A 0.000,B 0.000,C 90.000,E1 152.922} C_DIS
LIN {X 0.050,Y -161.362,Z 482.830,A 0.000,B 0.000,C 90.000,E1 149.331} C_DIS
LIN {X 0.062,Y -165.565,Z 482.810,A 0.000,B 0.000,C 90.000,E1 145.801} C_DIS
LIN {X -0.054,Y -170.482,Z 482.791,A 0.000,B 0.000,C 90.000,E1 142.351} C_DIS
LIN {X 0.095,Y -175.363,Z 482.772,A 0.000,B 0.000,C 90.000,E1 138.852} C_DIS
LIN {X -0.042,Y -180.987,Z 482.753,A 0.000,B 0.000,C 90.000,E1 135.486} C_DIS
LIN {X -0.055,Y -186.413,Z 482.734,A 0.000,B 0.000,C 90.000,E1 132.123} C_DIS
LIN {X -0.116,Y -191.041,Z 482.720,A 0.000,B 0.000,C 90.000,E1 129.644} C_DIS
LIN {X -0.116,Y -193.495,Z 482.712,A 0.000,B 0.000,C 90.000,E1 128.177} C_DIS
LIN {X -0.030,Y -290.585,Z 482.712,A 0.000,B 0.000,C 90.000,E1 128.141} C_DIS
LIN {X -0.060,Y -296.092,Z 482.711,A 0.000,B 0.000,C 90.000,E1 127.971} C_DIS
LIN {X 0.019,Y -299.041,Z 482.710,A 0.000,B 0.000,C 90.000,E1 127.729} C_DIS
LIN {X -0.027,Y -302.787,Z 482.707,A 0.000,B 0.000,C 90.000,E1 127.282} C_DIS
LIN {X -0.005,Y -304.668,Z 482.705,A 0.000,B 0.000,C 90.000,E1 126.950} C_DIS
LIN {X -0.044,Y -306.141,Z 482.703,A 0.000,B 0.000,C 90.000,E1 126.629} C_DIS
LIN {X 0.005,Y -308.271,Z 482.700,A 0.000,B 0.000,C 90.000,E1 125.964} C_DIS
LIN {X -0.181,Y -318.545,Z 482.682,A 0.000,B 0.000,C 90.000,E1 122.752} C_DIS
LIN {X -0.113,Y -329.129,Z 482.666,A 0.000,B 0.000,C 90.000,E1 119.873} C_DIS
LIN {X -0.073,Y -341.089,Z 482.650,A 0.000,B 0.000,C 90.000,E1 117.052} C_DIS
LIN {X 0.157,Y -354.525,Z 482.635,A 0.000,B 0.000,C 90.000,E1 114.259} C_DIS
LIN {X -0.062,Y -367.813,Z 482.622,A 0.000,B 0.000,C 90.000,E1 111.897} C_DIS
LIN {X -0.227,Y -382.462,Z 482.609,A 0.000,B 0.000,C 90.000,E1 109.577} C_DIS
LIN {X -0.157,Y -398.581,Z 482.596,A 0.000,B 0.000,C 90.000,E1 107.275} C_DIS
LIN {X 0.085,Y -416.289,Z 482.583,A 0.000,B 0.000,C 90.000,E1 105.009} C_DIS
LIN {X 0.211,Y -435.653,Z 482.571,A 0.000,B 0.000,C 90.000,E1 102.827} C_DIS
LIN {X 0.027,Y -455.904,Z 482.560,A 0.000,B 0.000,C 90.000,E1 100.838} C_DIS
LIN {X 0.187,Y -476.687,Z 482.550,A 0.000,B 0.000,C 90.000,E1 98.973} C_DIS
LIN {X -0.083,Y -481.803,Z 482.548,A 0.000,B 0.000,C 90.000,E1 98.568} C_DIS
LIN {X 0.003,Y -483.695,Z 482.546,A 0.000,B 0.000,C 90.000,E1 98.341} C_DIS
LIN {X -0.115,Y -485.352,Z 482.545,A 0.000,B 0.000,C 90.000,E1 98.106} C_DIS
LIN {X 0.246,Y -486.593,Z 482.544,A 0.000,B 0.000,C 90.000,E1 97.814} C_DIS
LIN {X -0.044,Y -488.115,Z 482.541,A 0.000,B 0.000,C 90.000,E1 97.352} C_DIS
LIN {X 0.158,Y -488.580,Z 482.538,A 0.000,B 0.000,C 90.000,E1 96.834} C_DIS
LIN {X -0.116,Y -488.067,Z 482.535,A 0.000,B 0.000,C 90.000,E1 96.372} C_DIS
LIN {X 0.098,Y -486.491,Z 482.533,A 0.000,B 0.000,C 90.000,E1 95.853} C_DIS
LIN {X -0.064,Y -485.218,Z 482.531,A 0.000,B 0.000,C 90.000,E1 95.625} C_DIS
LIN {X -0.176,Y -483.519,Z 482.530,A 0.000,B 0.000,C 90.000,E1 95.391} C_DIS
LIN {X -0.188,Y -471.414,Z 482.522,A 0.000,B 0.000,C 90.000,E1 93.898} C_DIS
LIN {X 0.063,Y -456.086,Z 482.510,A 0.000,B 0.000,C 90.000,E1 91.835} C_DIS
LIN {X -0.027,Y -442.447,Z 482.499,A 0.000,B 0.000,C 90.000,E1 89.771} C_DIS
LIN {X -0.136,Y -430.960,Z 482.488,A 0.000,B 0.000,C 90.000,E1 87.936} C_DIS
LIN {X 0.190,Y -416.384,Z 482.475,A 0.000,B 0.000,C 90.000,E1 85.469} C_DIS
LIN {X 0.167,Y -402.173,Z 482.461,A 0.000,B 0.000,C 90.000,E1 82.996} C_DIS
LIN {X -0.180,Y -391.229,Z 482.450,A 0.000,B 0.000,C 90.000,E1 81.084} C_DIS
LIN {X 0.049,Y -381.864,Z 482.441,A 0.000,B 0.000,C 90.000,E1 79.342} C_DIS
LIN {X -0.124,Y -366.477,Z 482.425,A 0.000,B 0.000,C 90.000,E1 76.464} C_DIS
LIN {X -0.149,Y -356.400,Z 482.413,A 0.000,B 0.000,C 90.000,E1 74.393} C_DIS
LIN {X 0.066,Y -346.149,Z 482.400,A 0.000,B 0.000,C 90.000,E1 71.945} C_DIS
LIN {X -0.097,Y -334.674,Z 482.383,A 0.000,B 0.000,C 90.000,E1 68.901} C_DIS
LIN {X 0.043,Y -322.904,Z 482.364,A 0.000,B 0.000,C 90.000,E1 65.433} C_DIS
LIN {X 0.124,Y -314.607,Z 482.349,A 0.000,B 0.000,C 90.000,E1 62.871} C_DIS
LIN {X -0.124,Y -306.373,Z 482.335,A 0.000,B 0.000,C 90.000,E1 60.333} C_DIS
LIN {X 0.145,Y -298.342,Z 482.320,A 0.000,B 0.000,C 90.000,E1 57.661} C_DIS
LIN {X 0.012,Y -288.765,Z 482.302,A 0.000,B 0.000,C 90.000,E1 54.356} C_DIS
LIN {X -0.095,Y -283.285,Z 482.291,A 0.000,B 0.000,C 90.000,E1 52.351} C_DIS
LIN {X 0.048,Y -277.686,Z 482.279,A 0.000,B 0.000,C 90.000,E1 50.275} C_DIS
LIN {X -0.126,Y -271.678,Z 482.268,A 0.000,B 0.000,C 90.000,E1 48.243} C_DIS
LIN {X -0.049,Y -265.292,Z 482.256,A 0.000,B 0.000,C 90.000,E1 46.134} C_DIS
LIN {X -0.104,Y -258.606,Z 482.244,A 0.000,B 0.000,C 90.000,E1 44.028} C_DIS
LIN {X -0.059,Y -248.560,Z 482.227,A 0.000,B 0.000,C 90.000,E1 40.782} C_DIS
LIN {X 0.118,Y -238.937,Z 482.208,A 0.000,B 0.000,C 90.000,E1 37.443} C_DIS
LIN {X 0.020,Y -230.938,Z 482.192,A 0.000,B 0.000,C 90.000,E1 34.485} C_DIS
LIN {X -0.018,Y -223.785,Z 482.175,A 0.000,B 0.000,C 90.000,E1 31.465} C_DIS
LIN {X 0.103,Y -217.571,Z 482.158,A 0.000,B 0.000,C 90.000,E1 28.359} C_DIS
LIN {X -0.043,Y -212.135,Z 482.140,A 0.000,B 0.000,C 90.000,E1 25.283} C_DIS
LIN {X -0.015,Y -206.395,Z 482.118,A 0.000,B 0.000,C 90.000,E1 21.334} C_DIS
LIN {X 0.033,Y -201.707,Z 482.096,A 0.000,B 0.000,C 90.000,E1 17.330} C_DIS
LIN {X 0.036,Y -197.963,Z 482.074,A 0.000,B 0.000,C 90.000,E1 13.300} C_DIS
LIN {X -0.088,Y -194.468,Z 482.042,A 0.000,B 0.000,C 90.000,E1 7.644} C_DIS
LIN {X 0.049,Y -195.331,Z 481.947,A 0.000,B 0.000,C 90.000,E1 350.500} C_DIS
LIN {X -0.057,Y -198.949,Z 481.920,A 0.000,B 0.000,C 90.000,E1 345.644} C_DIS
LIN {X 0.016,Y -202.857,Z 481.898,A 0.000,B 0.000,C 90.000,E1 341.583} C_DIS
LIN {X -0.029,Y -207.803,Z 481.875,A 0.000,B 0.000,C 90.000,E1 337.592} C_DIS
LIN {X -0.060,Y -213.424,Z 481.853,A 0.000,B 0.000,C 90.000,E1 333.640} C_DIS
LIN {X -0.118,Y -219.756,Z 481.832,A 0.000,B 0.000,C 90.000,E1 329.744} C_DIS
LIN {X -0.104,Y -226.630,Z 481.810,A 0.000,B 0.000,C 90.000,E1 325.881} C_DIS
LIN {X -0.050,Y -234.281,Z 481.789,A 0.000,B 0.000,C 90.000,E1 322.065} C_DIS
LIN {X -0.053,Y -242.675,Z 481.768,A 0.000,B 0.000,C 90.000,E1 318.324} C_DIS
LIN {X 0.000,Y -251.282,Z 481.750,A 0.000,B 0.000,C 90.000,E1 315.000} C_DIS
LIN {X -0.026,Y -260.970,Z 481.732,A 0.000,B 0.000,C 90.000,E1 311.757} C_DIS
LIN {X 0.108,Y -271.620,Z 481.714,A 0.000,B 0.000,C 90.000,E1 308.543} C_DIS
LIN {X 0.042,Y -283.319,Z 481.697,A 0.000,B 0.000,C 90.000,E1 305.438} C_DIS
LIN {X -0.116,Y -295.817,Z 481.680,A 0.000,B 0.000,C 90.000,E1 302.418} C_DIS
LIN {X -0.011,Y -307.561,Z 481.665,A 0.000,B 0.000,C 90.000,E1 299.745} C_DIS
LIN {X 0.025,Y -318.539,Z 481.653,A 0.000,B 0.000,C 90.000,E1 297.462} C_DIS
LIN {X 0.065,Y -336.181,Z 481.635,A 0.000,B 0.000,C 90.000,E1 294.283} C_DIS
LIN {X -0.134,Y -349.867,Z 481.623,A 0.000,B 0.000,C 90.000,E1 292.153} C_DIS
LIN {X -0.178,Y -369.347,Z 481.608,A 0.000,B 0.000,C 90.000,E1 289.450} C_DIS
LIN {X -0.178,Y -385.898,Z 481.597,A 0.000,B 0.000,C 90.000,E1 287.402} C_DIS
LIN {X -0.158,Y -410.787,Z 481.581,A 0.000,B 0.000,C 90.000,E1 284.592} C_DIS
LIN {X -0.199,Y -425.967,Z 481.572,A 0.000,B 0.000,C 90.000,E1 283.008} C_DIS
LIN {X 0.019,Y -438.485,Z 481.565,A 0.000,B 0.000,C 90.000,E1 281.658} C_DIS
LIN {X 0.033,Y -448.190,Z 481.559,A 0.000,B 0.000,C 90.000,E1 280.602} C_DIS
LIN {X -0.210,Y -454.944,Z 481.555,A 0.000,B 0.000,C 90.000,E1 279.849} C_DIS
LIN {X 0.127,Y -461.143,Z 481.550,A 0.000,B 0.000,C 90.000,E1 279.029} C_DIS
LIN {X -0.005,Y -466.760,Z 481.546,A 0.000,B 0.000,C 90.000,E1 278.276} C_DIS
LIN {X -0.159,Y -471.826,Z 481.542,A 0.000,B 0.000,C 90.000,E1 277.530} C_DIS
LIN {X -0.199,Y -476.364,Z 481.538,A 0.000,B 0.000,C 90.000,E1 276.777} C_DIS
LIN {X -0.211,Y -480.360,Z 481.533,A 0.000,B 0.000,C 90.000,E1 276.024} C_DIS
LIN {X 0.247,Y -483.746,Z 481.529,A 0.000,B 0.000,C 90.000,E1 275.220} C_DIS
LIN {X -0.229,Y -486.498,Z 481.525,A 0.000,B 0.000,C 90.000,E1 274.531} C_DIS
LIN {X -0.042,Y -487.899,Z 481.522,A 0.000,B 0.000,C 90.000,E1 274.012} C_DIS
LIN {X 0.123,Y -489.045,Z 481.520,A 0.000,B 0.000,C 90.000,E1 273.498} C_DIS
LIN {X -0.161,Y -489.807,Z 481.517,A 0.000,B 0.000,C 90.000,E1 273.037} C_DIS
LIN {X 0.024,Y -490.251,Z 481.514,A 0.000,B 0.000,C 90.000,E1 272.522} C_DIS
LIN {X 0.216,Y -490.353,Z 481.511,A 0.000,B 0.000,C 90.000,E1 272.007} C_DIS
LIN {X -0.063,Y -489.983,Z 481.509,A 0.000,B 0.000,C 90.000,E1 271.547} C_DIS
LIN {X 0.133,Y -489.196,Z 481.506,A 0.000,B 0.000,C 90.000,E1 271.031} C_DIS
LIN {X -0.162,Y -487.887,Z 481.503,A 0.000,B 0.000,C 90.000,E1 270.573} C_DIS
LIN {X 0.029,Y -486.015,Z 481.500,A 0.000,B 0.000,C 90.000,E1 270.057} C_DIS
LIN {X 0.211,Y -483.458,Z 481.498,A 0.000,B 0.000,C 90.000,E1 269.542} C_DIS
LIN {X 0.051,Y -481.936,Z 481.496,A 0.000,B 0.000,C 90.000,E1 269.312} C_DIS
LIN {X 0.203,Y -478.171,Z 481.493,A 0.000,B 0.000,C 90.000,E1 268.797} C_DIS
LIN {X -0.140,Y -473.517,Z 481.491,A 0.000,B 0.000,C 90.000,E1 268.339} C_DIS
LIN {X 0.153,Y -467.920,Z 481.488,A 0.000,B 0.000,C 90.000,E1 267.822} C_DIS
LIN {X -0.109,Y -461.682,Z 481.486,A 0.000,B 0.000,C 90.000,E1 267.421} C_DIS
LIN {X 0.135,Y -454.997,Z 481.484,A 0.000,B 0.000,C 90.000,E1 267.020} C_DIS
LIN {X -0.044,Y -448.225,Z 481.482,A 0.000,B 0.000,C 90.000,E1 266.731} C_DIS
LIN {X 0.121,Y -441.060,Z 481.480,A 0.000,B 0.000,C 90.000,E1 266.445} C_DIS
LIN {X -0.197,Y -433.233,Z 481.479,A 0.000,B 0.000,C 90.000,E1 266.274} C_DIS
LIN {X -0.078,Y -424.814,Z 481.478,A 0.000,B 0.000,C 90.000,E1 266.102} C_DIS
LIN {X -0.031,Y -414.750,Z 481.478,A 0.000,B 0.000,C 90.000,E1 265.988} C_DIS
LIN {X 0.140,Y -408.594,Z 481.478,A 0.000,B 0.000,C 90.000,E1 265.931} C_DIS
LIN {X 0.040,Y -180.917,Z 481.477,A 0.000,B 0.000,C 90.000,E1 265.927} C_DIS
LIN {X 0.070,Y -180.840,Z 481.472,A 0.000,B 0.000,C 90.000,E1 264.894} C_DIS
LIN {X -0.033,Y -178.882,Z 481.443,A 0.000,B 0.000,C 90.000,E1 259.690} C_DIS
LIN {X 0.042,Y -175.925,Z 481.414,A 0.000,B 0.000,C 90.000,E1 254.574} C_DIS
LIN {X -0.013,Y -175.364,Z 481.410,A 0.000,B 0.000,C 90.000,E1 253.740} C_DIS
LIN {X 0.046,Y -172.142,Z 481.386,A 0.000,B 0.000,C 90.000,E1 249.444} C_DIS
LIN {X 0.023,Y -171.606,Z 481.381,A 0.000,B 0.000,C 90.000,E1 248.592} C_DIS
LIN {X 0.012,Y -167.829,Z 481.357,A 0.000,B 0.000,C 90.000,E1 244.280} C_DIS
LIN {X 0.029,Y -166.554,Z 481.347,A 0.000,B 0.000,C 90.000,E1 242.538} C_DIS
LIN {X -0.061,Y -162.549,Z 481.323,A 0.000,B 0.000,C 90.000,E1 238.201} C_DIS
LIN {X 0.000,Y -161.228,Z 481.313,A 0.000,B 0.000,C 90.000,E1 236.421} C_DIS
LIN {X 0.034,Y -157.233,Z 481.289,A 0.000,B 0.000,C 90.000,E1 231.984} C_DIS
LIN {X 0.057,Y -155.958,Z 481.279,A 0.000,B 0.000,C 90.000,E1 230.194} C_DIS
LIN {X 0.016,Y -152.212,Z 481.254,A 0.000,B 0.000,C 90.000,E1 225.729} C_DIS
LIN {X 0.036,Y -150.456,Z 481.239,A 0.000,B 0.000,C 90.000,E1 223.014} C_DIS
LIN {X 0.063,Y -147.181,Z 481.214,A 0.000,B 0.000,C 90.000,E1 218.463} C_DIS
LIN {X 0.029,Y -145.199,Z 481.194,A 0.000,B 0.000,C 90.000,E1 214.818} C_DIS
LIN {X -0.060,Y -142.337,Z 481.163,A 0.000,B 0.000,C 90.000,E1 209.333} C_DIS
LIN {X -0.007,Y -141.726,Z 481.153,A 0.000,B 0.000,C 90.000,E1 207.462} C_DIS
LIN {X -0.024,Y -139.480,Z 481.116,A 0.000,B 0.000,C 90.000,E1 200.972} C_DIS
LIN {X -0.035,Y -138.979,Z 481.101,A 0.000,B 0.000,C 90.000,E1 198.181} C_DIS
LIN {X -0.051,Y -138.332,Z 481.054,A 0.000,B 0.000,C 90.000,E1 189.782} C_DIS
LIN {X -0.050,Y -139.430,Z 481.008,A 0.000,B 0.000,C 90.000,E1 181.375} C_DIS
LIN {X 0.003,Y -141.358,Z 480.971,A 0.000,B 0.000,C 90.000,E1 174.837} C_DIS
LIN {X -0.021,Y -142.711,Z 480.956,A 0.000,B 0.000,C 90.000,E1 172.064} C_DIS
LIN {X -0.062,Y -145.087,Z 480.930,A 0.000,B 0.000,C 90.000,E1 167.465} C_DIS
LIN {X 0.075,Y -147.711,Z 480.910,A 0.000,B 0.000,C 90.000,E1 163.740} C_DIS
LIN {X 0.016,Y -150.367,Z 480.890,A 0.000,B 0.000,C 90.000,E1 160.115} C_DIS
LIN {X 0.035,Y -153.793,Z 480.869,A 0.000,B 0.000,C 90.000,E1 156.485} C_DIS
LIN {X -0.046,Y -157.206,Z 480.849,A 0.000,B 0.000,C 90.000,E1 152.922} C_DIS
LIN {X 0.036,Y -161.370,Z 480.830,A 0.000,B 0.000,C 90.000,E1 149.331} C_DIS
LIN {X 0.047,Y -165.572,Z 480.810,A 0.000,B 0.000,C 90.000,E1 145.801} C_DIS
LIN {X -0.070,Y -170.490,Z 480.791,A 0.000,B 0.000,C 90.000,E1 142.351} C_DIS
LIN {X 0.079,Y -175.371,Z 480.772,A 0.000,B 0.000,C 90.000,E1 138.852} C_DIS
LIN {X -0.057,Y -180.995,Z 480.753,A 0.000,B 0.000,C 90.000,E1 135.486} C_DIS
LIN {X 0.067,Y -186.423,Z 480.734,A 0.000,B 0.000,C 90.000,E1 132.081} C_DIS
LIN {X 0.015,Y -191.050,Z 480.720,A 0.000,B 0.000,C 90.000,E1 129.600} C_DIS
LIN {X -0.007,Y -193.579,Z 480.712,A 0.000,B 0.000,C 90.000,E1 128.096} C_DIS
LIN {X -0.047,Y -290.898,Z 480.712,A 0.000,B 0.000,C 90.000,E1 128.096} C_DIS
LIN {X -0.153,Y -292.365,Z 480.711,A 0.000,B 0.000,C 90.000,E1 128.096} C_DIS
LIN {X 0.097,Y -295.439,Z 480.711,A 0.000,B 0.000,C 90.000,E1 127.935} C_DIS
LIN {X -0.024,Y -298.719,Z 480.710,A 0.000,B 0.000,C 90.000,E1 127.729} C_DIS
LIN {X -0.069,Y -302.394,Z 480.707,A 0.000,B 0.000,C 90.000,E1 127.317} C_DIS
LIN {X -0.031,Y -304.318,Z 480.706,A 0.000,B 0.000,C 90.000,E1 126.996} C_DIS
LIN {X 0.068,Y -305.832,Z 480.704,A 0.000,B 0.000,C 90.000,E1 126.664} C_DIS
LIN {X -0.156,Y -307.088,Z 480.702,A 0.000,B 0.000,C 90.000,E1 126.377} C_DIS
LIN {X 0.116,Y -318.341,Z 480.682,A 0.000,B 0.000,C 90.000,E1 122.752} C_DIS
LIN {X -0.097,Y -328.901,Z 480.666,A 0.000,B 0.000,C 90.000,E1 119.922} C_DIS
LIN {X 0.077,Y -340.834,Z 480.651,A 0.000,B 0.000,C 90.000,E1 117.078} C_DIS
LIN {X -0.003,Y -354.242,Z 480.635,A 0.000,B 0.000,C 90.000,E1 114.335} C_DIS
LIN {X -0.089,Y -367.501,Z 480.622,A 0.000,B 0.000,C 90.000,E1 111.950} C_DIS
LIN {X 0.091,Y -382.122,Z 480.609,A 0.000,B 0.000,C 90.000,E1 109.577} C_DIS
LIN {X 0.166,Y -398.209,Z 480.596,A 0.000,B 0.000,C 90.000,E1 107.275} C_DIS
LIN {X 0.011,Y -415.883,Z 480.584,A 0.000,B 0.000,C 90.000,E1 105.064} C_DIS
LIN {X 0.112,Y -435.219,Z 480.572,A 0.000,B 0.000,C 90.000,E1 102.883} C_DIS
LIN {X -0.109,Y -455.458,Z 480.560,A 0.000,B 0.000,C 90.000,E1 100.894} C_DIS
LIN {X 0.013,Y -476.231,Z 480.550,A 0.000,B 0.000,C 90.000,E1 99.029} C_DIS
LIN {X 0.211,Y -481.437,Z 480.548,A 0.000,B 0.000,C 90.000,E1 98.568} C_DIS
LIN {X -0.183,Y -483.458,Z 480.547,A 0.000,B 0.000,C 90.000,E1 98.398} C_DIS
LIN {X 0.177,Y -485.215,Z 480.545,A 0.000,B 0.000,C 90.000,E1 98.106} C_DIS
LIN {X 0.056,Y -486.534,Z 480.544,A 0.000,B 0.000,C 90.000,E1 97.871} C_DIS
LIN {X 0.248,Y -488.177,Z 480.541,A 0.000,B 0.000,C 90.000,E1 97.352} C_DIS
LIN {X -0.035,Y -488.746,Z 480.538,A 0.000,B 0.000,C 90.000,E1 96.891} C_DIS
LIN {X 0.177,Y -488.333,Z 480.536,A 0.000,B 0.000,C 90.000,E1 96.372} C_DIS
LIN {X -0.095,Y -486.875,Z 480.533,A 0.000,B 0.000,C 90.000,E1 95.910} C_DIS
LIN {X 0.229,Y -485.675,Z 480.531,A 0.000,B 0.000,C 90.000,E1 95.625} C_DIS
LIN {X 0.115,Y -484.072,Z 480.530,A 0.000,B 0.000,C 90.000,E1 95.391} C_DIS
LIN {X 0.106,Y -471.997,Z 480.522,A 0.000,B 0.000,C 90.000,E1 93.898} C_DIS
LIN {X -0.097,Y -456.602,Z 480.510,A 0.000,B 0.000,C 90.000,E1 91.892} C_DIS
LIN {X -0.170,Y -442.903,Z 480.499,A 0.000,B 0.000,C 90.000,E1 89.828} C_DIS
LIN {X 0.165,Y -431.407,Z 480.489,A 0.000,B 0.000,C 90.000,E1 87.936} C_DIS
LIN {X 0.076,Y -416.825,Z 480.475,A 0.000,B 0.000,C 90.000,E1 85.527} C_DIS
LIN {X 0.071,Y -402.625,Z 480.461,A 0.000,B 0.000,C 90.000,E1 83.053} C_DIS
LIN {X 0.123,Y -391.678,Z 480.451,A 0.000,B 0.000,C 90.000,E1 81.084} C_DIS
LIN {X -0.023,Y -382.331,Z 480.441,A 0.000,B 0.000,C 90.000,E1 79.398} C_DIS
LIN {X 0.183,Y -366.944,Z 480.425,A 0.000,B 0.000,C 90.000,E1 76.464} C_DIS
LIN {X 0.158,Y -356.828,Z 480.413,A 0.000,B 0.000,C 90.000,E1 74.393} C_DIS
LIN {X 0.046,Y -346.535,Z 480.400,A 0.000,B 0.000,C 90.000,E1 72.000} C_DIS
LIN {X -0.108,Y -333.883,Z 480.381,A 0.000,B 0.000,C 90.000,E1 68.646} C_DIS
LIN {X 0.057,Y -323.154,Z 480.364,A 0.000,B 0.000,C 90.000,E1 65.485} C_DIS
LIN {X 0.008,Y -314.795,Z 480.350,A 0.000,B 0.000,C 90.000,E1 62.948} C_DIS
LIN {X -0.086,Y -306.535,Z 480.335,A 0.000,B 0.000,C 90.000,E1 60.383} C_DIS
LIN {X 0.033,Y -298.461,Z 480.321,A 0.000,B 0.000,C 90.000,E1 57.740} C_DIS
LIN {X 0.070,Y -288.840,Z 480.302,A 0.000,B 0.000,C 90.000,E1 54.402} C_DIS
LIN {X -0.030,Y -283.362,Z 480.291,A 0.000,B 0.000,C 90.000,E1 52.396} C_DIS
LIN {X -0.060,Y -277.756,Z 480.280,A 0.000,B 0.000,C 90.000,E1 50.356} C_DIS
LIN {X 0.154,Y -271.735,Z 480.268,A 0.000,B 0.000,C 90.000,E1 48.243} C_DIS
LIN {X -0.148,Y -265.382,Z 480.257,A 0.000,B 0.000,C 90.000,E1 46.215} C_DIS
LIN {X 0.172,Y -258.721,Z 480.245,A 0.000,B 0.000,C 90.000,E1 44.028} C_DIS
LIN {X -0.157,Y -249.777,Z 480.229,A 0.000,B 0.000,C 90.000,E1 41.229} C_DIS
LIN {X 0.073,Y -241.163,Z 480.213,A 0.000,B 0.000,C 90.000,E1 38.257} C_DIS
LIN {X -0.019,Y -233.021,Z 480.196,A 0.000,B 0.000,C 90.000,E1 35.311} C_DIS
LIN {X -0.005,Y -225.623,Z 480.179,A 0.000,B 0.000,C 90.000,E1 32.291} C_DIS
LIN {X 0.085,Y -219.163,Z 480.162,A 0.000,B 0.000,C 90.000,E1 29.205} C_DIS
LIN {X 0.072,Y -213.521,Z 480.145,A 0.000,B 0.000,C 90.000,E1 26.104} C_DIS
LIN {X -0.049,Y -207.537,Z 480.123,A 0.000,B 0.000,C 90.000,E1 22.206} C_DIS
LIN {X -0.086,Y -202.611,Z 480.101,A 0.000,B 0.000,C 90.000,E1 18.236} C_DIS
LIN {X 0.001,Y -198.636,Z 480.079,A 0.000,B 0.000,C 90.000,E1 14.189} C_DIS
LIN {X -0.003,Y -195.261,Z 480.052,A 0.000,B 0.000,C 90.000,E1 9.321} C_DIS
LIN {X 0.093,Y -192.837,Z 480.015,A 0.000,B 0.000,C 90.000,E1 2.751} C_DIS
LIN {X 0.064,Y -194.357,Z 479.956,A 0.000,B 0.000,C 90.000,E1 352.129} C_DIS
LIN {X 0.072,Y -197.454,Z 479.929,A 0.000,B 0.000,C 90.000,E1 347.229} C_DIS
LIN {X 0.092,Y -201.863,Z 479.902,A 0.000,B 0.000,C 90.000,E1 342.362} C_DIS
LIN {X 0.063,Y -206.587,Z 479.880,A 0.000,B 0.000,C 90.000,E1 338.358} C_DIS
LIN {X -0.013,Y -212.089,Z 479.858,A 0.000,B 0.000,C 90.000,E1 334.409} C_DIS
LIN {X 0.081,Y -218.305,Z 479.836,A 0.000,B 0.000,C 90.000,E1 330.461} C_DIS
LIN {X -0.061,Y -225.037,Z 479.815,A 0.000,B 0.000,C 90.000,E1 326.628} C_DIS
LIN {X -0.003,Y -232.537,Z 479.793,A 0.000,B 0.000,C 90.000,E1 322.798} C_DIS
LIN {X -0.060,Y -240.817,Z 479.772,A 0.000,B 0.000,C 90.000,E1 319.057} C_DIS
LIN {X -0.050,Y -249.182,Z 479.754,A 0.000,B 0.000,C 90.000,E1 315.729} C_DIS
LIN {X 0.035,Y -258.636,Z 479.736,A 0.000,B 0.000,C 90.000,E1 312.447} C_DIS
LIN {X -0.036,Y -270.334,Z 479.716,A 0.000,B 0.000,C 90.000,E1 308.910} C_DIS
LIN {X -0.028,Y -283.298,Z 479.697,A 0.000,B 0.000,C 90.000,E1 305.438} C_DIS
LIN {X -0.038,Y -297.257,Z 479.678,A 0.000,B 0.000,C 90.000,E1 302.054} C_DIS
LIN {X -0.015,Y -310.607,Z 479.662,A 0.000,B 0.000,C 90.000,E1 299.077} C_DIS
LIN {X 0.084,Y -321.939,Z 479.649,A 0.000,B 0.000,C 90.000,E1 296.796} C_DIS
LIN {X 0.085,Y -340.000,Z 479.631,A 0.000,B 0.000,C 90.000,E1 293.643} C_DIS
LIN {X -0.170,Y -354.075,Z 479.619,A 0.000,B 0.000,C 90.000,E1 291.535} C_DIS
LIN {X 0.168,Y -371.712,Z 479.606,A 0.000,B 0.000,C 90.000,E1 289.087} C_DIS
LIN {X -0.141,Y -388.320,Z 479.595,A 0.000,B 0.000,C 90.000,E1 287.094} C_DIS
LIN {X -0.057,Y -413.331,Z 479.579,A 0.000,B 0.000,C 90.000,E1 284.300} C_DIS
LIN {X -0.030,Y -428.676,Z 479.571,A 0.000,B 0.000,C 90.000,E1 282.703} C_DIS
LIN {X 0.151,Y -441.128,Z 479.563,A 0.000,B 0.000,C 90.000,E1 281.366} C_DIS
LIN {X 0.093,Y -448.159,Z 479.559,A 0.000,B 0.000,C 90.000,E1 280.602} C_DIS
LIN {X -0.148,Y -454.932,Z 479.555,A 0.000,B 0.000,C 90.000,E1 279.849} C_DIS
LIN {X 0.189,Y -461.127,Z 479.550,A 0.000,B 0.000,C 90.000,E1 279.029} C_DIS
LIN {X 0.058,Y -466.776,Z 479.546,A 0.000,B 0.000,C 90.000,E1 278.276} C_DIS
LIN {X -0.095,Y -471.868,Z 479.542,A 0.000,B 0.000,C 90.000,E1 277.530} C_DIS
LIN {X -0.135,Y -476.416,Z 479.538,A 0.000,B 0.000,C 90.000,E1 276.777} C_DIS
LIN {X -0.145,Y -480.419,Z 479.533,A 0.000,B 0.000,C 90.000,E1 276.024} C_DIS
LIN {X -0.168,Y -483.828,Z 479.529,A 0.000,B 0.000,C 90.000,E1 275.277} C_DIS
LIN {X -0.162,Y -486.596,Z 479.525,A 0.000,B 0.000,C 90.000,E1 274.531} C_DIS
LIN {X 0.026,Y -488.020,Z 479.522,A 0.000,B 0.000,C 90.000,E1 274.012} C_DIS
LIN {X 0.193,Y -489.150,Z 479.520,A 0.000,B 0.000,C 90.000,E1 273.498} C_DIS
LIN {X -0.091,Y -489.929,Z 479.517,A 0.000,B 0.000,C 90.000,E1 273.037} C_DIS
LIN {X 0.095,Y -490.380,Z 479.514,A 0.000,B 0.000,C 90.000,E1 272.522} C_DIS
LIN {X -0.202,Y -490.446,Z 479.511,A 0.000,B 0.000,C 90.000,E1 272.064} C_DIS
LIN {X 0.008,Y -490.126,Z 479.509,A 0.000,B 0.000,C 90.000,E1 271.547} C_DIS
LIN {X 0.204,Y -489.333,Z 479.506,A 0.000,B 0.000,C 90.000,E1 271.031} C_DIS
LIN {X -0.088,Y -488.045,Z 479.503,A 0.000,B 0.000,C 90.000,E1 270.573} C_DIS
LIN {X 0.103,Y -486.182,Z 479.500,A 0.000,B 0.000,C 90.000,E1 270.057} C_DIS
LIN {X -0.200,Y -483.653,Z 479.498,A 0.000,B 0.000,C 90.000,E1 269.599} C_DIS
LIN {X -0.034,Y -480.373,Z 479.495,A 0.000,B 0.000,C 90.000,E1 269.083} C_DIS
LIN {X 0.111,Y -476.175,Z 479.492,A 0.000,B 0.000,C 90.000,E1 268.568} C_DIS
LIN {X -0.066,Y -473.754,Z 479.491,A 0.000,B 0.000,C 90.000,E1 268.339} C_DIS
LIN {X 0.230,Y -468.138,Z 479.488,A 0.000,B 0.000,C 90.000,E1 267.822} C_DIS
LIN {X 0.214,Y -465.022,Z 479.487,A 0.000,B 0.000,C 90.000,E1 267.593} C_DIS
LIN {X 0.169,Y -458.419,Z 479.485,A 0.000,B 0.000,C 90.000,E1 267.192} C_DIS
LIN {X -0.232,Y -451.764,Z 479.483,A 0.000,B 0.000,C 90.000,E1 266.906} C_DIS
LIN {X 0.221,Y -444.853,Z 479.481,A 0.000,B 0.000,C 90.000,E1 266.560} C_DIS
LIN {X 0.100,Y -437.310,Z 479.480,A 0.000,B 0.000,C 90.000,E1 266.331} C_DIS
LIN {X -0.049,Y -428.611,Z 479.479,A 0.000,B 0.000,C 90.000,E1 266.159} C_DIS
LIN {X -0.149,Y -419.493,Z 479.478,A 0.000,B 0.000,C 90.000,E1 266.045} C_DIS
LIN {X -0.215,Y -411.033,Z 479.478,A 0.000,B 0.000,C 90.000,E1 265.988} C_DIS
LIN {X 0.143,Y -407.852,Z 479.477,A 0.000,B 0.000,C 90.000,E1 265.927} C_DIS
LIN {X 0.028,Y -180.917,Z 479.477,A 0.000,B 0.000,C 90.000,E1 265.927} C_DIS
LIN {X 0.057,Y -180.840,Z 479.472,A 0.000,B 0.000,C 90.000,E1 264.894} C_DIS
LIN {X -0.046,Y -178.880,Z 479.443,A 0.000,B 0.000,C 90.000,E1 259.690} C_DIS
LIN {X 0.031,Y -175.924,Z 479.414,A 0.000,B 0.000,C 90.000,E1 254.574} C_DIS
LIN {X -0.024,Y -175.360,Z 479.410,A 0.000,B 0.000,C 90.000,E1 253.740} C_DIS
LIN {X 0.035,Y -172.140,Z 479.386,A 0.000,B 0.000,C 90.000,E1 249.444} C_DIS
LIN {X 0.011,Y -171.603,Z 479.381,A 0.000,B 0.000,C 90.000,E1 248.592} C_DIS
LIN {X 0.001,Y -167.826,Z 479.357,A 0.000,B 0.000,C 90.000,E1 244.280} C_DIS
LIN {X 0.018,Y -166.550,Z 479.347,A 0.000,B 0.000,C 90.000,E1 242.538} C_DIS
LIN {X -0.072,Y -162.546,Z 479.323,A 0.000,B 0.000,C 90.000,E1 238.201} C_DIS
LIN {X -0.011,Y -161.224,Z 479.313,A 0.000,B 0.000,C 90.000,E1 236.421} C_DIS
LIN {X 0.023,Y -157.230,Z 479.289,A 0.000,B 0.000,C 90.000,E1 231.984} C_DIS
LIN {X 0.047,Y -155.955,Z 479.279,A 0.000,B 0.000,C 90.000,E1 230.194} C_DIS
LIN {X 0.006,Y -152.209,Z 479.254,A 0.000,B 0.000,C 90.000,E1 225.729} C_DIS
LIN {X 0.026,Y -150.454,Z 479.239,A 0.000,B 0.000,C 90.000,E1 223.014} C_DIS
LIN {X 0.053,Y -147.179,Z 479.214,A 0.000,B 0.000,C 90.000,E1 218.463} C_DIS
LIN {X 0.019,Y -145.196,Z 479.193,A 0.000,B 0.000,C 90.000,E1 214.818} C_DIS
LIN {X 0.054,Y -142.335,Z 479.163,A 0.000,B 0.000,C 90.000,E1 209.283} C_DIS
LIN {X -0.017,Y -141.724,Z 479.153,A 0.000,B 0.000,C 90.000,E1 207.462} C_DIS
LIN {X -0.035,Y -139.479,Z 479.116,A 0.000,B 0.000,C 90.000,E1 200.972} C_DIS
LIN {X -0.046,Y -138.977,Z 479.101,A 0.000,B 0.000,C 90.000,E1 198.181} C_DIS
LIN {X 0.075,Y -138.332,Z 479.054,A 0.000,B 0.000,C 90.000,E1 189.726} C_DIS
LIN {X -0.060,Y -139.431,Z 479.008,A 0.000,B 0.000,C 90.000,E1 181.375} C_DIS
LIN {X 0.019,Y -140.956,Z 478.976,A 0.000,B 0.000,C 90.000,E1 175.755} C_DIS
LIN {X -0.031,Y -142.713,Z 478.956,A 0.000,B 0.000,C 90.000,E1 172.064} C_DIS
LIN {X 0.069,Y -145.089,Z 478.930,A 0.000,B 0.000,C 90.000,E1 167.409} C_DIS
LIN {X 0.064,Y -147.714,Z 478.910,A 0.000,B 0.000,C 90.000,E1 163.740} C_DIS
LIN {X 0.006,Y -150.371,Z 478.890,A 0.000,B 0.000,C 90.000,E1 160.115} C_DIS
LIN {X 0.024,Y -153.798,Z 478.869,A 0.000,B 0.000,C 90.000,E1 156.485} C_DIS
LIN {X 0.084,Y -157.210,Z 478.849,A 0.000,B 0.000,C 90.000,E1 152.871} C_DIS
LIN {X 0.025,Y -161.374,Z 478.830,A 0.000,B 0.000,C 90.000,E1 149.331} C_DIS
LIN {X 0.036,Y -165.577,Z 478.810,A 0.000,B 0.000,C 90.000,E1 145.801} C_DIS
LIN {X 0.023,Y -170.496,Z 478.791,A 0.000,B 0.000,C 90.000,E1 142.316} C_DIS
LIN {X 0.068,Y -175.376,Z 478.772,A 0.000,B 0.000,C 90.000,E1 138.852} C_DIS
LIN {X -0.069,Y -181.001,Z 478.753,A 0.000,B 0.000,C 90.000,E1 135.486} C_DIS
LIN {X 0.055,Y -186.428,Z 478.734,A 0.000,B 0.000,C 90.000,E1 132.081} C_DIS
LIN {X 0.124,Y -191.055,Z 478.720,A 0.000,B 0.000,C 90.000,E1 129.564} C_DIS
LIN {X 0.101,Y -193.663,Z 478.711,A 0.000,B 0.000,C 90.000,E1 128.016} C_DIS
LIN {X 0.117,Y -290.755,Z 478.711,A 0.000,B 0.000,C 90.000,E1 128.016} C_DIS
LIN {X 0.077,Y -294.580,Z 478.711,A 0.000,B 0.000,C 90.000,E1 127.935} C_DIS
LIN {X -0.176,Y -297.604,Z 478.710,A 0.000,B 0.000,C 90.000,E1 127.810} C_DIS
LIN {X -0.113,Y -301.256,Z 478.708,A 0.000,B 0.000,C 90.000,E1 127.443} C_DIS
LIN {X -0.010,Y -304.822,Z 478.705,A 0.000,B 0.000,C 90.000,E1 126.870} C_DIS
LIN {X 0.003,Y -306.324,Z 478.703,A 0.000,B 0.000,C 90.000,E1 126.537} C_DIS
LIN {X -0.050,Y -307.510,Z 478.701,A 0.000,B 0.000,C 90.000,E1 126.217} C_DIS
LIN {X -0.006,Y -317.691,Z 478.683,A 0.000,B 0.000,C 90.000,E1 122.959} C_DIS
LIN {X 0.044,Y -328.167,Z 478.667,A 0.000,B 0.000,C 90.000,E1 120.079} C_DIS
LIN {X 0.067,Y -340.009,Z 478.651,A 0.000,B 0.000,C 90.000,E1 117.257} C_DIS
LIN {X -0.044,Y -353.320,Z 478.636,A 0.000,B 0.000,C 90.000,E1 114.515} C_DIS
LIN {X 0.043,Y -366.485,Z 478.623,A 0.000,B 0.000,C 90.000,E1 112.099} C_DIS
LIN {X -0.011,Y -381.004,Z 478.610,A 0.000,B 0.000,C 90.000,E1 109.758} C_DIS
LIN {X 0.032,Y -396.983,Z 478.597,A 0.000,B 0.000,C 90.000,E1 107.457} C_DIS
LIN {X -0.159,Y -414.538,Z 478.585,A 0.000,B 0.000,C 90.000,E1 105.245} C_DIS
LIN {X -0.113,Y -433.769,Z 478.572,A 0.000,B 0.000,C 90.000,E1 103.063} C_DIS
LIN {X 0.094,Y -453.968,Z 478.561,A 0.000,B 0.000,C 90.000,E1 101.007} C_DIS
LIN {X 0.050,Y -474.705,Z 478.551,A 0.000,B 0.000,C 90.000,E1 99.151} C_DIS
LIN {X -0.105,Y -482.398,Z 478.547,A 0.000,B 0.000,C 90.000,E1 98.511} C_DIS
LIN {X -0.057,Y -484.323,Z 478.546,A 0.000,B 0.000,C 90.000,E1 98.276} C_DIS
LIN {X -0.076,Y -485.796,Z 478.545,A 0.000,B 0.000,C 90.000,E1 98.049} C_DIS
LIN {X -0.191,Y -487.006,Z 478.543,A 0.000,B 0.000,C 90.000,E1 97.814} C_DIS
LIN {X 0.113,Y -487.890,Z 478.542,A 0.000,B 0.000,C 90.000,E1 97.530} C_DIS
LIN {X -0.165,Y -488.825,Z 478.539,A 0.000,B 0.000,C 90.000,E1 97.068} C_DIS
LIN {X 0.047,Y -488.766,Z 478.536,A 0.000,B 0.000,C 90.000,E1 96.549} C_DIS
LIN {X -0.221,Y -487.702,Z 478.534,A 0.000,B 0.000,C 90.000,E1 96.087} C_DIS
LIN {X 0.155,Y -486.744,Z 478.532,A 0.000,B 0.000,C 90.000,E1 95.796} C_DIS
LIN {X -0.004,Y -485.442,Z 478.531,A 0.000,B 0.000,C 90.000,E1 95.568} C_DIS
LIN {X 0.198,Y -481.729,Z 478.528,A 0.000,B 0.000,C 90.000,E1 95.049} C_DIS
LIN {X 0.098,Y -459.955,Z 478.513,A 0.000,B 0.000,C 90.000,E1 92.293} C_DIS
LIN {X 0.125,Y -449.228,Z 478.504,A 0.000,B 0.000,C 90.000,E1 90.745} C_DIS
LIN {X -0.129,Y -436.005,Z 478.493,A 0.000,B 0.000,C 90.000,E1 88.682} C_DIS
LIN {X -0.095,Y -421.294,Z 478.479,A 0.000,B 0.000,C 90.000,E1 86.274} C_DIS
LIN {X 0.026,Y -407.013,Z 478.466,A 0.000,B 0.000,C 90.000,E1 83.799} C_DIS
LIN {X 0.193,Y -394.519,Z 478.453,A 0.000,B 0.000,C 90.000,E1 81.546} C_DIS
LIN {X 0.109,Y -382.039,Z 478.441,A 0.000,B 0.000,C 90.000,E1 79.285} C_DIS
LIN {X -0.065,Y -366.686,Z 478.424,A 0.000,B 0.000,C 90.000,E1 76.408} C_DIS
LIN {X -0.087,Y -356.613,Z 478.413,A 0.000,B 0.000,C 90.000,E1 74.338} C_DIS
LIN {X -0.202,Y -346.335,Z 478.400,A 0.000,B 0.000,C 90.000,E1 71.945} C_DIS
LIN {X -0.038,Y -334.806,Z 478.382,A 0.000,B 0.000,C 90.000,E1 68.847} C_DIS
LIN {X -0.029,Y -323.968,Z 478.365,A 0.000,B 0.000,C 90.000,E1 65.717} C_DIS
LIN {X -0.045,Y -315.526,Z 478.351,A 0.000,B 0.000,C 90.000,E1 63.179} C_DIS
LIN {X 0.010,Y -307.224,Z 478.337,A 0.000,B 0.000,C 90.000,E1 60.589} C_DIS
LIN {X -0.111,Y -299.110,Z 478.322,A 0.000,B 0.000,C 90.000,E1 57.995} C_DIS
LIN {X 0.027,Y -289.397,Z 478.304,A 0.000,B 0.000,C 90.000,E1 54.642} C_DIS
LIN {X -0.069,Y -283.914,Z 478.292,A 0.000,B 0.000,C 90.000,E1 52.637} C_DIS
LIN {X 0.085,Y -278.294,Z 478.281,A 0.000,B 0.000,C 90.000,E1 50.561} C_DIS
LIN {X -0.074,Y -272.335,Z 478.270,A 0.000,B 0.000,C 90.000,E1 48.528} C_DIS
LIN {X 0.020,Y -266.007,Z 478.258,A 0.000,B 0.000,C 90.000,E1 46.419} C_DIS
LIN {X -0.016,Y -259.405,Z 478.246,A 0.000,B 0.000,C 90.000,E1 44.312} C_DIS
LIN {X 0.024,Y -250.495,Z 478.230,A 0.000,B 0.000,C 90.000,E1 41.434} C_DIS
LIN {X -0.092,Y -241.820,Z 478.214,A 0.000,B 0.000,C 90.000,E1 38.543} C_DIS
LIN {X -0.027,Y -233.648,Z 478.198,A 0.000,B 0.000,C 90.000,E1 35.564} C_DIS
LIN {X -0.005,Y -226.201,Z 478.181,A 0.000,B 0.000,C 90.000,E1 32.546} C_DIS
LIN {X -0.013,Y -219.659,Z 478.164,A 0.000,B 0.000,C 90.000,E1 29.489} C_DIS
LIN {X 0.093,Y -213.962,Z 478.147,A 0.000,B 0.000,C 90.000,E1 26.360} C_DIS
LIN {X -0.014,Y -207.882,Z 478.125,A 0.000,B 0.000,C 90.000,E1 22.461} C_DIS
LIN {X -0.034,Y -202.879,Z 478.103,A 0.000,B 0.000,C 90.000,E1 18.489} C_DIS
LIN {X -0.072,Y -198.821,Z 478.080,A 0.000,B 0.000,C 90.000,E1 14.481} C_DIS
LIN {X -0.070,Y -195.352,Z 478.053,A 0.000,B 0.000,C 90.000,E1 9.613} C_DIS
LIN {X 0.049,Y -192.795,Z 478.017,A 0.000,B 0.000,C 90.000,E1 3.037} C_DIS
LIN {X 0.058,Y -194.234,Z 477.956,A 0.000,B 0.000,C 90.000,E1 352.129} C_DIS
LIN {X 0.061,Y -197.315,Z 477.929,A 0.000,B 0.000,C 90.000,E1 347.229} C_DIS
LIN {X 0.076,Y -201.724,Z 477.902,A 0.000,B 0.000,C 90.000,E1 342.362} C_DIS
LIN {X 0.041,Y -206.424,Z 477.880,A 0.000,B 0.000,C 90.000,E1 338.358} C_DIS
LIN {X -0.041,Y -211.937,Z 477.858,A 0.000,B 0.000,C 90.000,E1 334.409} C_DIS
LIN {X 0.048,Y -218.171,Z 477.836,A 0.000,B 0.000,C 90.000,E1 330.461} C_DIS
LIN {X -0.099,Y -224.892,Z 477.814,A 0.000,B 0.000,C 90.000,E1 326.628} C_DIS
LIN {X 0.094,Y -232.404,Z 477.793,A 0.000,B 0.000,C 90.000,E1 322.763} C_DIS
LIN {X 0.071,Y -240.682,Z 477.772,A 0.000,B 0.000,C 90.000,E1 319.013} C_DIS
LIN {X 0.079,Y -248.080,Z 477.756,A 0.000,B 0.000,C 90.000,E1 316.053} C_DIS
LIN {X 0.136,Y -257.432,Z 477.738,A 0.000,B 0.000,C 90.000,E1 312.771} C_DIS
LIN {X -0.170,Y -269.055,Z 477.718,A 0.000,B 0.000,C 90.000,E1 309.277} C_DIS
LIN {X 0.020,Y -281.925,Z 477.699,A 0.000,B 0.000,C 90.000,E1 305.758} C_DIS
LIN {X 0.144,Y -295.811,Z 477.680,A 0.000,B 0.000,C 90.000,E1 302.339} C_DIS
LIN {X -0.012,Y -307.573,Z 477.665,A 0.000,B 0.000,C 90.000,E1 299.716} C_DIS
LIN {X -0.065,Y -320.257,Z 477.651,A 0.000,B 0.000,C 90.000,E1 297.129} C_DIS
LIN {X 0.019,Y -338.140,Z 477.633,A 0.000,B 0.000,C 90.000,E1 293.951} C_DIS
LIN {X 0.171,Y -352.037,Z 477.621,A 0.000,B 0.000,C 90.000,E1 291.770} C_DIS
LIN {X -0.006,Y -369.454,Z 477.608,A 0.000,B 0.000,C 90.000,E1 289.396} C_DIS
LIN {X 0.138,Y -388.344,Z 477.595,A 0.000,B 0.000,C 90.000,E1 287.040} C_DIS
LIN {X 0.133,Y -410.807,Z 477.581,A 0.000,B 0.000,C 90.000,E1 284.537} C_DIS
LIN {X -0.070,Y -428.734,Z 477.571,A 0.000,B 0.000,C 90.000,E1 282.703} C_DIS
LIN {X -0.134,Y -441.015,Z 477.563,A 0.000,B 0.000,C 90.000,E1 281.422} C_DIS
LIN {X 0.096,Y -448.202,Z 477.559,A 0.000,B 0.000,C 90.000,E1 280.602} C_DIS
LIN {X -0.145,Y -454.975,Z 477.555,A 0.000,B 0.000,C 90.000,E1 279.849} C_DIS
LIN {X 0.193,Y -461.200,Z 477.550,A 0.000,B 0.000,C 90.000,E1 279.029} C_DIS
LIN {X 0.062,Y -466.836,Z 477.546,A 0.000,B 0.000,C 90.000,E1 278.276} C_DIS
LIN {X -0.089,Y -471.939,Z 477.542,A 0.000,B 0.000,C 90.000,E1 277.530} C_DIS
LIN {X -0.129,Y -476.496,Z 477.538,A 0.000,B 0.000,C 90.000,E1 276.777} C_DIS
LIN {X -0.139,Y -480.507,Z 477.533,A 0.000,B 0.000,C 90.000,E1 276.024} C_DIS
LIN {X -0.161,Y -483.947,Z 477.529,A 0.000,B 0.000,C 90.000,E1 275.277} C_DIS
LIN {X -0.153,Y -486.702,Z 477.525,A 0.000,B 0.000,C 90.000,E1 274.531} C_DIS
LIN {X 0.036,Y -488.129,Z 477.522,A 0.000,B 0.000,C 90.000,E1 274.012} C_DIS
LIN {X 0.203,Y -489.269,Z 477.520,A 0.000,B 0.000,C 90.000,E1 273.498} C_DIS
LIN {X -0.081,Y -490.056,Z 477.517,A 0.000,B 0.000,C 90.000,E1 273.037} C_DIS
LIN {X 0.105,Y -490.512,Z 477.514,A 0.000,B 0.000,C 90.000,E1 272.522} C_DIS
LIN {X -0.191,Y -490.595,Z 477.511,A 0.000,B 0.000,C 90.000,E1 272.064} C_DIS
LIN {X 0.021,Y -490.272,Z 477.509,A 0.000,B 0.000,C 90.000,E1 271.547} C_DIS
LIN {X 0.218,Y -489.472,Z 477.506,A 0.000,B 0.000,C 90.000,E1 271.031} C_DIS
LIN {X -0.074,Y -488.151,Z 477.503,A 0.000,B 0.000,C 90.000,E1 270.573} C_DIS
LIN {X 0.118,Y -486.305,Z 477.500,A 0.000,B 0.000,C 90.000,E1 270.057} C_DIS
LIN {X -0.184,Y -483.784,Z 477.498,A 0.000,B 0.000,C 90.000,E1 269.599} C_DIS
LIN {X -0.019,Y -480.528,Z 477.495,A 0.000,B 0.000,C 90.000,E1 269.083} C_DIS
LIN {X 0.128,Y -476.295,Z 477.492,A 0.000,B 0.000,C 90.000,E1 268.568} C_DIS
LIN {X -0.049,Y -473.886,Z 477.491,A 0.000,B 0.000,C 90.000,E1 268.339} C_DIS
LIN {X -0.202,Y -468.300,Z 477.488,A 0.000,B 0.000,C 90.000,E1 267.879} C_DIS
LIN {X 0.026,Y -462.125,Z 477.486,A 0.000,B 0.000,C 90.000,E1 267.421} C_DIS
LIN {X -0.196,Y -455.502,Z 477.484,A 0.000,B 0.000,C 90.000,E1 267.078} C_DIS
LIN {X 0.065,Y -448.715,Z 477.482,A 0.000,B 0.000,C 90.000,E1 266.731} C_DIS
LIN {X 0.214,Y -441.583,Z 477.480,A 0.000,B 0.000,C 90.000,E1 266.445} C_DIS
LIN {X -0.156,Y -433.713,Z 477.479,A 0.000,B 0.000,C 90.000,E1 266.274} C_DIS
LIN {X -0.079,Y -424.901,Z 477.478,A 0.000,B 0.000,C 90.000,E1 266.102} C_DIS
LIN {X -0.037,Y -414.666,Z 477.478,A 0.000,B 0.000,C 90.000,E1 265.988} C_DIS
LIN {X 0.134,Y -409.521,Z 477.478,A 0.000,B 0.000,C 90.000,E1 265.931} C_DIS
LIN {X 0.037,Y -180.917,Z 477.477,A 0.000,B 0.000,C 90.000,E1 265.927} C_DIS
LIN {X 0.067,Y -180.841,Z 477.472,A 0.000,B 0.000,C 90.000,E1 264.894} C_DIS
LIN {X -0.037,Y -178.882,Z 477.443,A 0.000,B 0.000,C 90.000,E1 259.690} C_DIS
LIN {X 0.039,Y -175.924,Z 477.414,A 0.000,B 0.000,C 90.000,E1 254.574} C_DIS
LIN {X -0.015,Y -175.363,Z 477.410,A 0.000,B 0.000,C 90.000,E1 253.740} C_DIS
LIN {X 0.043,Y -172.141,Z 477.386,A 0.000,B 0.000,C 90.000,E1 249.444} C_DIS
LIN {X 0.021,Y -171.605,Z 477.381,A 0.000,B 0.000,C 90.000,E1 248.592} C_DIS
LIN {X 0.009,Y -167.828,Z 477.357,A 0.000,B 0.000,C 90.000,E1 244.280} C_DIS
LIN {X 0.026,Y -166.553,Z 477.347,A 0.000,B 0.000,C 90.000,E1 242.538} C_DIS
LIN {X -0.063,Y -162.548,Z 477.323,A 0.000,B 0.000,C 90.000,E1 238.201} C_DIS
LIN {X -0.004,Y -161.227,Z 477.313,A 0.000,B 0.000,C 90.000,E1 236.421} C_DIS
LIN {X 0.032,Y -157.233,Z 477.289,A 0.000,B 0.000,C 90.000,E1 231.984} C_DIS
LIN {X 0.055,Y -155.956,Z 477.279,A 0.000,B 0.000,C 90.000,E1 230.194} C_DIS
LIN {X 0.013,Y -152.211,Z 477.254,A 0.000,B 0.000,C 90.000,E1 225.729} C_DIS
LIN {X 0.034,Y -150.455,Z 477.239,A 0.000,B 0.000,C 90.000,E1 223.014} C_DIS
LIN {X 0.060,Y -147.181,Z 477.214,A 0.000,B 0.000,C 90.000,E1 218.463} C_DIS
LIN {X 0.027,Y -145.199,Z 477.193,A 0.000,B 0.000,C 90.000,E1 214.818} C_DIS
LIN {X 0.061,Y -142.336,Z 477.163,A 0.000,B 0.000,C 90.000,E1 209.283} C_DIS
LIN {X -0.010,Y -141.726,Z 477.153,A 0.000,B 0.000,C 90.000,E1 207.462} C_DIS
LIN {X -0.028,Y -139.480,Z 477.116,A 0.000,B 0.000,C 90.000,E1 200.972} C_DIS
LIN {X -0.038,Y -138.978,Z 477.101,A 0.000,B 0.000,C 90.000,E1 198.181} C_DIS
LIN {X -0.053,Y -138.332,Z 477.054,A 0.000,B 0.000,C 90.000,E1 189.782} C_DIS
LIN {X -0.053,Y -139.430,Z 477.008,A 0.000,B 0.000,C 90.000,E1 181.375} C_DIS
LIN {X 0.001,Y -141.359,Z 476.971,A 0.000,B 0.000,C 90.000,E1 174.837} C_DIS
LIN {X -0.024,Y -142.712,Z 476.956,A 0.000,B 0.000,C 90.000,E1 172.064} C_DIS
LIN {X -0.065,Y -145.088,Z 476.930,A 0.000,B 0.000,C 90.000,E1 167.465} C_DIS
LIN {X 0.072,Y -147.712,Z 476.910,A 0.000,B 0.000,C 90.000,E1 163.740} C_DIS
LIN {X 0.013,Y -150.368,Z 476.890,A 0.000,B 0.000,C 90.000,E1 160.115} C_DIS
LIN {X 0.032,Y -153.795,Z 476.869,A 0.000,B 0.000,C 90.000,E1 156.485} C_DIS
LIN {X -0.048,Y -157.207,Z 476.849,A 0.000,B 0.000,C 90.000,E1 152.922} C_DIS
LIN {X 0.033,Y -161.370,Z 476.830,A 0.000,B 0.000,C 90.000,E1 149.331} C_DIS
LIN {X 0.044,Y -165.573,Z 476.810,A 0.000,B 0.000,C 90.000,E1 145.801} C_DIS
LIN {X -0.072,Y -170.492,Z 476.791,A 0.000,B 0.000,C 90.000,E1 142.351} C_DIS
LIN {X 0.076,Y -175.372,Z 476.772,A 0.000,B 0.000,C 90.000,E1 138.852} C_DIS
LIN {X -0.060,Y -180.996,Z 476.753,A 0.000,B 0.000,C 90.000,E1 135.486} C_DIS
LIN {X 0.064,Y -186.424,Z 476.734,A 0.000,B 0.000,C 90.000,E1 132.081} C_DIS
LIN {X 0.011,Y -191.051,Z 476.720,A 0.000,B 0.000,C 90.000,E1 129.600} C_DIS
LIN {X -0.068,Y -193.751,Z 476.711,A 0.000,B 0.000,C 90.000,E1 128.016} C_DIS
LIN {X -0.132,Y -290.762,Z 476.711,A 0.000,B 0.000,C 90.000,E1 128.016} C_DIS
LIN {X 0.091,Y -293.180,Z 476.711,A 0.000,B 0.000,C 90.000,E1 127.935} C_DIS
LIN {X -0.002,Y -296.494,Z 476.710,A 0.000,B 0.000,C 90.000,E1 127.810} C_DIS
LIN {X 0.078,Y -299.888,Z 476.709,A 0.000,B 0.000,C 90.000,E1 127.523} C_DIS
LIN {X -0.054,Y -303.553,Z 476.706,A 0.000,B 0.000,C 90.000,E1 127.076} C_DIS
LIN {X -0.047,Y -305.360,Z 476.704,A 0.000,B 0.000,C 90.000,E1 126.744} C_DIS
LIN {X 0.145,Y -306.777,Z 476.702,A 0.000,B 0.000,C 90.000,E1 126.377} C_DIS
LIN {X 0.132,Y -308.843,Z 476.699,A 0.000,B 0.000,C 90.000,E1 125.724} C_DIS
LIN {X 0.059,Y -319.213,Z 476.681,A 0.000,B 0.000,C 90.000,E1 122.498} C_DIS
LIN {X -0.126,Y -329.894,Z 476.665,A 0.000,B 0.000,C 90.000,E1 119.667} C_DIS
LIN {X 0.081,Y -341.957,Z 476.649,A 0.000,B 0.000,C 90.000,E1 116.821} C_DIS
LIN {X 0.032,Y -355.507,Z 476.634,A 0.000,B 0.000,C 90.000,E1 114.079} C_DIS
LIN {X -0.163,Y -368.902,Z 476.621,A 0.000,B 0.000,C 90.000,E1 111.716} C_DIS
LIN {X 0.187,Y -383.668,Z 476.608,A 0.000,B 0.000,C 90.000,E1 109.322} C_DIS
LIN {X 0.177,Y -399.914,Z 476.595,A 0.000,B 0.000,C 90.000,E1 107.040} C_DIS
LIN {X 0.067,Y -417.758,Z 476.582,A 0.000,B 0.000,C 90.000,E1 104.828} C_DIS
LIN {X -0.172,Y -437.233,Z 476.570,A 0.000,B 0.000,C 90.000,E1 102.703} C_DIS
LIN {X 0.181,Y -457.531,Z 476.559,A 0.000,B 0.000,C 90.000,E1 100.658} C_DIS
LIN {X 0.032,Y -481.005,Z 476.548,A 0.000,B 0.000,C 90.000,E1 98.624} C_DIS
LIN {X 0.107,Y -483.229,Z 476.547,A 0.000,B 0.000,C 90.000,E1 98.398} C_DIS
LIN {X 0.253,Y -484.918,Z 476.546,A 0.000,B 0.000,C 90.000,E1 98.163} C_DIS
LIN {X 0.070,Y -486.394,Z 476.544,A 0.000,B 0.000,C 90.000,E1 97.936} C_DIS
LIN {X -0.046,Y -487.494,Z 476.543,A 0.000,B 0.000,C 90.000,E1 97.701} C_DIS
LIN {X 0.155,Y -488.792,Z 476.540,A 0.000,B 0.000,C 90.000,E1 97.182} C_DIS
LIN {X -0.122,Y -489.065,Z 476.537,A 0.000,B 0.000,C 90.000,E1 96.720} C_DIS
LIN {X 0.095,Y -488.353,Z 476.535,A 0.000,B 0.000,C 90.000,E1 96.201} C_DIS
LIN {X -0.173,Y -486.536,Z 476.532,A 0.000,B 0.000,C 90.000,E1 95.739} C_DIS
LIN {X 0.152,Y -485.105,Z 476.530,A 0.000,B 0.000,C 90.000,E1 95.454} C_DIS
LIN {X 0.052,Y -477.223,Z 476.525,A 0.000,B 0.000,C 90.000,E1 94.473} C_DIS
LIN {X -0.221,Y -459.516,Z 476.512,A 0.000,B 0.000,C 90.000,E1 92.236} C_DIS
LIN {X -0.194,Y -448.824,Z 476.504,A 0.000,B 0.000,C 90.000,E1 90.688} C_DIS
LIN {X -0.011,Y -435.588,Z 476.492,A 0.000,B 0.000,C 90.000,E1 88.568} C_DIS
LIN {X 0.143,Y -419.286,Z 476.477,A 0.000,B 0.000,C 90.000,E1 85.869} C_DIS
LIN {X 0.211,Y -405.062,Z 476.463,A 0.000,B 0.000,C 90.000,E1 83.394} C_DIS
LIN {X -0.128,Y -394.156,Z 476.453,A 0.000,B 0.000,C 90.000,E1 81.489} C_DIS
LIN {X -0.143,Y -381.677,Z 476.440,A 0.000,B 0.000,C 90.000,E1 79.218} C_DIS
LIN {X -0.032,Y -366.365,Z 476.424,A 0.000,B 0.000,C 90.000,E1 76.297} C_DIS
LIN {X 0.026,Y -356.352,Z 476.412,A 0.000,B 0.000,C 90.000,E1 74.212} C_DIS
LIN {X -0.070,Y -344.886,Z 476.397,A 0.000,B 0.000,C 90.000,E1 71.511} C_DIS
LIN {X 0.053,Y -333.437,Z 476.380,A 0.000,B 0.000,C 90.000,E1 68.411} C_DIS
LIN {X -0.029,Y -324.744,Z 476.366,A 0.000,B 0.000,C 90.000,E1 65.921} C_DIS
LIN {X -0.035,Y -316.241,Z 476.352,A 0.000,B 0.000,C 90.000,E1 63.384} C_DIS
LIN {X 0.032,Y -307.892,Z 476.338,A 0.000,B 0.000,C 90.000,E1 60.795} C_DIS
LIN {X -0.076,Y -299.722,Z 476.323,A 0.000,B 0.000,C 90.000,E1 58.201} C_DIS
LIN {X 0.080,Y -289.933,Z 476.305,A 0.000,B 0.000,C 90.000,E1 54.848} C_DIS
LIN {X -0.131,Y -282.548,Z 476.290,A 0.000,B 0.000,C 90.000,E1 52.190} C_DIS
LIN {X 0.001,Y -276.880,Z 476.278,A 0.000,B 0.000,C 90.000,E1 50.114} C_DIS
LIN {X 0.018,Y -270.843,Z 476.267,A 0.000,B 0.000,C 90.000,E1 48.038} C_DIS
LIN {X -0.119,Y -264.462,Z 476.255,A 0.000,B 0.000,C 90.000,E1 45.972} C_DIS
LIN {X 0.005,Y -257.819,Z 476.243,A 0.000,B 0.000,C 90.000,E1 43.824} C_DIS
LIN {X 0.019,Y -248.959,Z 476.227,A 0.000,B 0.000,C 90.000,E1 40.943} C_DIS
LIN {X 0.007,Y -238.270,Z 476.207,A 0.000,B 0.000,C 90.000,E1 37.282} C_DIS
LIN {X -0.106,Y -230.406,Z 476.191,A 0.000,B 0.000,C 90.000,E1 34.326} C_DIS
LIN {X 0.029,Y -223.351,Z 476.174,A 0.000,B 0.000,C 90.000,E1 31.258} C_DIS
LIN {X 0.033,Y -217.182,Z 476.157,A 0.000,B 0.000,C 90.000,E1 28.180} C_DIS
LIN {X -0.026,Y -211.794,Z 476.139,A 0.000,B 0.000,C 90.000,E1 25.079} C_DIS
LIN {X 0.100,Y -206.052,Z 476.117,A 0.000,B 0.000,C 90.000,E1 21.099} C_DIS
LIN {X -0.053,Y -201.376,Z 476.095,A 0.000,B 0.000,C 90.000,E1 17.149} C_DIS
LIN {X -0.059,Y -197.649,Z 476.073,A 0.000,B 0.000,C 90.000,E1 13.119} C_DIS
LIN {X -0.011,Y -194.159,Z 476.041,A 0.000,B 0.000,C 90.000,E1 7.409} C_DIS
LIN {X -0.084,Y -193.728,Z 475.961,A 0.000,B 0.000,C 90.000,E1 352.989} C_DIS
LIN {X 0.029,Y -196.560,Z 475.934,A 0.000,B 0.000,C 90.000,E1 348.049} C_DIS
LIN {X -0.035,Y -200.770,Z 475.907,A 0.000,B 0.000,C 90.000,E1 343.196} C_DIS
LIN {X 0.028,Y -205.250,Z 475.884,A 0.000,B 0.000,C 90.000,E1 339.156} C_DIS
LIN {X 0.016,Y -210.622,Z 475.862,A 0.000,B 0.000,C 90.000,E1 335.177} C_DIS
LIN {X -0.042,Y -216.723,Z 475.840,A 0.000,B 0.000,C 90.000,E1 331.257} C_DIS
LIN {X -0.048,Y -223.353,Z 475.819,A 0.000,B 0.000,C 90.000,E1 327.375} C_DIS
LIN {X -0.035,Y -230.705,Z 475.797,A 0.000,B 0.000,C 90.000,E1 323.543} C_DIS
LIN {X 0.075,Y -238.832,Z 475.776,A 0.000,B 0.000,C 90.000,E1 319.747} C_DIS
LIN {X 0.053,Y -246.026,Z 475.760,A 0.000,B 0.000,C 90.000,E1 316.782} C_DIS
LIN {X 0.042,Y -255.159,Z 475.742,A 0.000,B 0.000,C 90.000,E1 313.500} C_DIS
LIN {X -0.049,Y -265.375,Z 475.724,A 0.000,B 0.000,C 90.000,E1 310.297} C_DIS
LIN {X -0.132,Y -276.605,Z 475.706,A 0.000,B 0.000,C 90.000,E1 307.156} C_DIS
LIN {X -0.029,Y -290.118,Z 475.687,A 0.000,B 0.000,C 90.000,E1 303.706} C_DIS
LIN {X 0.099,Y -303.121,Z 475.671,A 0.000,B 0.000,C 90.000,E1 300.669} C_DIS
LIN {X -0.125,Y -316.986,Z 475.654,A 0.000,B 0.000,C 90.000,E1 297.769} C_DIS
LIN {X -0.123,Y -327.251,Z 475.643,A 0.000,B 0.000,C 90.000,E1 295.848} C_DIS
LIN {X -0.091,Y -342.028,Z 475.630,A 0.000,B 0.000,C 90.000,E1 293.334} C_DIS
LIN {X 0.065,Y -358.417,Z 475.616,A 0.000,B 0.000,C 90.000,E1 290.865} C_DIS
LIN {X 0.053,Y -376.455,Z 475.603,A 0.000,B 0.000,C 90.000,E1 288.489} C_DIS
LIN {X -0.131,Y -398.081,Z 475.589,A 0.000,B 0.000,C 90.000,E1 285.953} C_DIS
LIN {X 0.094,Y -420.920,Z 475.575,A 0.000,B 0.000,C 90.000,E1 283.480} C_DIS
LIN {X 0.097,Y -433.510,Z 475.568,A 0.000,B 0.000,C 90.000,E1 282.187} C_DIS
LIN {X -0.066,Y -443.200,Z 475.562,A 0.000,B 0.000,C 90.000,E1 281.186} C_DIS
LIN {X -0.116,Y -452.514,Z 475.556,A 0.000,B 0.000,C 90.000,E1 280.141} C_DIS
LIN {X 0.207,Y -458.933,Z 475.552,A 0.000,B 0.000,C 90.000,E1 279.321} C_DIS
LIN {X 0.053,Y -464.825,Z 475.548,A 0.000,B 0.000,C 90.000,E1 278.568} C_DIS
LIN {X -0.048,Y -470.147,Z 475.543,A 0.000,B 0.000,C 90.000,E1 277.814} C_DIS
LIN {X -0.169,Y -474.928,Z 475.539,A 0.000,B 0.000,C 90.000,E1 277.068} C_DIS
LIN {X -0.184,Y -479.143,Z 475.535,A 0.000,B 0.000,C 90.000,E1 276.315} C_DIS
LIN {X -0.220,Y -482.812,Z 475.531,A 0.000,B 0.000,C 90.000,E1 275.568} C_DIS
LIN {X -0.048,Y -484.911,Z 475.528,A 0.000,B 0.000,C 90.000,E1 275.049} C_DIS
LIN {X 0.138,Y -486.699,Z 475.525,A 0.000,B 0.000,C 90.000,E1 274.531} C_DIS
LIN {X -0.160,Y -488.174,Z 475.522,A 0.000,B 0.000,C 90.000,E1 274.069} C_DIS
LIN {X 0.006,Y -489.297,Z 475.520,A 0.000,B 0.000,C 90.000,E1 273.555} C_DIS
LIN {X 0.212,Y -490.142,Z 475.517,A 0.000,B 0.000,C 90.000,E1 273.037} C_DIS
LIN {X -0.091,Y -490.611,Z 475.514,A 0.000,B 0.000,C 90.000,E1 272.579} C_DIS
LIN {X 0.103,Y -490.751,Z 475.512,A 0.000,B 0.000,C 90.000,E1 272.064} C_DIS
LIN {X -0.174,Y -490.409,Z 475.509,A 0.000,B 0.000,C 90.000,E1 271.604} C_DIS
LIN {X 0.024,Y -489.658,Z 475.506,A 0.000,B 0.000,C 90.000,E1 271.088} C_DIS
LIN {X 0.220,Y -488.376,Z 475.503,A 0.000,B 0.000,C 90.000,E1 270.573} C_DIS
LIN {X -0.074,Y -486.566,Z 475.501,A 0.000,B 0.000,C 90.000,E1 270.115} C_DIS
LIN {X 0.110,Y -484.076,Z 475.498,A 0.000,B 0.000,C 90.000,E1 269.599} C_DIS
LIN {X -0.205,Y -480.866,Z 475.495,A 0.000,B 0.000,C 90.000,E1 269.141} C_DIS
LIN {X -0.055,Y -476.745,Z 475.492,A 0.000,B 0.000,C 90.000,E1 268.625} C_DIS
LIN {X 0.085,Y -471.630,Z 475.490,A 0.000,B 0.000,C 90.000,E1 268.108} C_DIS
LIN {X 0.036,Y -468.797,Z 475.488,A 0.000,B 0.000,C 90.000,E1 267.879} C_DIS
LIN {X 0.210,Y -462.558,Z 475.486,A 0.000,B 0.000,C 90.000,E1 267.421} C_DIS
LIN {X -0.008,Y -456.020,Z 475.484,A 0.000,B 0.000,C 90.000,E1 267.078} C_DIS
LIN {X 0.232,Y -449.363,Z 475.482,A 0.000,B 0.000,C 90.000,E1 266.731} C_DIS
LIN {X -0.086,Y -442.275,Z 475.480,A 0.000,B 0.000,C 90.000,E1 266.502} C_DIS
LIN {X -0.028,Y -434.594,Z 475.479,A 0.000,B 0.000,C 90.000,E1 266.274} C_DIS
LIN {X 0.025,Y -425.925,Z 475.478,A 0.000,B 0.000,C 90.000,E1 266.102} C_DIS
LIN {X -0.122,Y -413.368,Z 475.478,A 0.000,B 0.000,C 90.000,E1 265.988} C_DIS
LIN {X 0.099,Y -406.275,Z 475.477,A 0.000,B 0.000,C 90.000,E1 265.927} C_DIS
LIN {X 0.020,Y -180.918,Z 475.477,A 0.000,B 0.000,C 90.000,E1 265.927} C_DIS
LIN {X -0.062,Y -180.872,Z 475.472,A 0.000,B 0.000,C 90.000,E1 265.065} C_DIS
LIN {X -0.005,Y -178.988,Z 475.444,A 0.000,B 0.000,C 90.000,E1 259.982} C_DIS
LIN {X 0.007,Y -177.968,Z 475.435,A 0.000,B 0.000,C 90.000,E1 258.285} C_DIS
LIN {X 0.026,Y -175.612,Z 475.411,A 0.000,B 0.000,C 90.000,E1 254.031} C_DIS
LIN {X 0.038,Y -172.334,Z 475.388,A 0.000,B 0.000,C 90.000,E1 249.752} C_DIS
LIN {X 0.016,Y -171.811,Z 475.383,A 0.000,B 0.000,C 90.000,E1 248.901} C_DIS
LIN {X 0.023,Y -170.274,Z 475.373,A 0.000,B 0.000,C 90.000,E1 247.177} C_DIS
LIN {X -0.040,Y -166.815,Z 475.349,A 0.000,B 0.000,C 90.000,E1 242.871} C_DIS
LIN {X 0.017,Y -162.796,Z 475.325,A 0.000,B 0.000,C 90.000,E1 238.486} C_DIS
LIN {X 0.077,Y -161.484,Z 475.315,A 0.000,B 0.000,C 90.000,E1 236.707} C_DIS
LIN {X -0.007,Y -157.480,Z 475.291,A 0.000,B 0.000,C 90.000,E1 232.316} C_DIS
LIN {X 0.050,Y -155.496,Z 475.276,A 0.000,B 0.000,C 90.000,E1 229.622} C_DIS
LIN {X -0.018,Y -151.801,Z 475.251,A 0.000,B 0.000,C 90.000,E1 225.162} C_DIS
LIN {X -0.005,Y -150.011,Z 475.236,A 0.000,B 0.000,C 90.000,E1 222.447} C_DIS
LIN {X 0.026,Y -146.837,Z 475.211,A 0.000,B 0.000,C 90.000,E1 217.890} C_DIS
LIN {X 0.012,Y -145.418,Z 475.195,A 0.000,B 0.000,C 90.000,E1 215.152} C_DIS
LIN {X 0.048,Y -142.846,Z 475.170,A 0.000,B 0.000,C 90.000,E1 210.541} C_DIS
LIN {X -0.023,Y -141.460,Z 475.149,A 0.000,B 0.000,C 90.000,E1 206.873} C_DIS
LIN {X 0.017,Y -139.375,Z 475.113,A 0.000,B 0.000,C 90.000,E1 200.355} C_DIS
LIN {X -0.042,Y -138.825,Z 475.098,A 0.000,B 0.000,C 90.000,E1 197.583} C_DIS
LIN {X 0.047,Y -138.352,Z 475.056,A 0.000,B 0.000,C 90.000,E1 190.074} C_DIS
LIN {X 0.021,Y -139.531,Z 475.004,A 0.000,B 0.000,C 90.000,E1 180.745} C_DIS
LIN {X -0.026,Y -141.210,Z 474.973,A 0.000,B 0.000,C 90.000,E1 175.179} C_DIS
LIN {X 0.074,Y -142.584,Z 474.958,A 0.000,B 0.000,C 90.000,E1 172.356} C_DIS
LIN {X 0.028,Y -144.880,Z 474.932,A 0.000,B 0.000,C 90.000,E1 167.757} C_DIS
LIN {X -0.018,Y -147.508,Z 474.912,A 0.000,B 0.000,C 90.000,E1 164.102} C_DIS
LIN {X 0.057,Y -150.100,Z 474.891,A 0.000,B 0.000,C 90.000,E1 160.423} C_DIS
LIN {X 0.070,Y -153.456,Z 474.871,A 0.000,B 0.000,C 90.000,E1 156.794} C_DIS
LIN {X -0.079,Y -157.820,Z 474.846,A 0.000,B 0.000,C 90.000,E1 152.359} C_DIS
LIN {X -0.048,Y -162.102,Z 474.827,A 0.000,B 0.000,C 90.000,E1 148.791} C_DIS
LIN {X -0.023,Y -166.303,Z 474.807,A 0.000,B 0.000,C 90.000,E1 145.261} C_DIS
LIN {X -0.026,Y -171.320,Z 474.788,A 0.000,B 0.000,C 90.000,E1 141.778} C_DIS
LIN {X 0.008,Y -176.220,Z 474.768,A 0.000,B 0.000,C 90.000,E1 138.324} C_DIS
LIN {X 0.002,Y -180.498,Z 474.754,A 0.000,B 0.000,C 90.000,E1 135.769} C_DIS
LIN {X -0.017,Y -185.902,Z 474.736,A 0.000,B 0.000,C 90.000,E1 132.405} C_DIS
LIN {X 0.044,Y -190.528,Z 474.722,A 0.000,B 0.000,C 90.000,E1 129.886} C_DIS
LIN {X 0.026,Y -193.843,Z 474.711,A 0.000,B 0.000,C 90.000,E1 127.935} C_DIS
LIN {X -0.008,Y -291.760,Z 474.711,A 0.000,B 0.000,C 90.000,E1 127.935} C_DIS
LIN {X 0.079,Y -293.241,Z 474.711,A 0.000,B 0.000,C 90.000,E1 127.890} C_DIS
LIN {X 0.085,Y -298.005,Z 474.709,A 0.000,B 0.000,C 90.000,E1 127.649} C_DIS
LIN {X -0.094,Y -300.618,Z 474.708,A 0.000,B 0.000,C 90.000,E1 127.443} C_DIS
LIN {X 0.132,Y -304.396,Z 474.705,A 0.000,B 0.000,C 90.000,E1 126.870} C_DIS
LIN {X -0.103,Y -306.042,Z 474.703,A 0.000,B 0.000,C 90.000,E1 126.583} C_DIS
LIN {X 0.089,Y -307.340,Z 474.701,A 0.000,B 0.000,C 90.000,E1 126.217} C_DIS
LIN {X -0.065,Y -318.662,Z 474.681,A 0.000,B 0.000,C 90.000,E1 122.673} C_DIS
LIN {X 0.001,Y -329.275,Z 474.666,A 0.000,B 0.000,C 90.000,E1 119.795} C_DIS
LIN {X -0.109,Y -341.259,Z 474.650,A 0.000,B 0.000,C 90.000,E1 117.001} C_DIS
LIN {X 0.127,Y -354.730,Z 474.635,A 0.000,B 0.000,C 90.000,E1 114.207} C_DIS
LIN {X -0.082,Y -368.047,Z 474.621,A 0.000,B 0.000,C 90.000,E1 111.844} C_DIS
LIN {X -0.108,Y -382.729,Z 474.608,A 0.000,B 0.000,C 90.000,E1 109.504} C_DIS
LIN {X -0.155,Y -398.884,Z 474.596,A 0.000,B 0.000,C 90.000,E1 107.221} C_DIS
LIN {X 0.100,Y -416.630,Z 474.583,A 0.000,B 0.000,C 90.000,E1 104.954} C_DIS
LIN {X -0.188,Y -436.038,Z 474.571,A 0.000,B 0.000,C 90.000,E1 102.827} C_DIS
LIN {X 0.090,Y -456.303,Z 474.560,A 0.000,B 0.000,C 90.000,E1 100.782} C_DIS
LIN {X -0.187,Y -477.099,Z 474.550,A 0.000,B 0.000,C 90.000,E1 98.973} C_DIS
LIN {X 0.022,Y -482.257,Z 474.547,A 0.000,B 0.000,C 90.000,E1 98.511} C_DIS
LIN {X 0.124,Y -484.255,Z 474.546,A 0.000,B 0.000,C 90.000,E1 98.276} C_DIS
LIN {X 0.157,Y -485.788,Z 474.545,A 0.000,B 0.000,C 90.000,E1 98.049} C_DIS
LIN {X 0.043,Y -487.090,Z 474.543,A 0.000,B 0.000,C 90.000,E1 97.814} C_DIS
LIN {X -0.137,Y -488.050,Z 474.542,A 0.000,B 0.000,C 90.000,E1 97.587} C_DIS
LIN {X 0.070,Y -489.115,Z 474.539,A 0.000,B 0.000,C 90.000,E1 97.068} C_DIS
LIN {X -0.203,Y -489.172,Z 474.537,A 0.000,B 0.000,C 90.000,E1 96.606} C_DIS
LIN {X 0.016,Y -488.236,Z 474.534,A 0.000,B 0.000,C 90.000,E1 96.087} C_DIS
LIN {X -0.250,Y -486.140,Z 474.531,A 0.000,B 0.000,C 90.000,E1 95.625} C_DIS
LIN {X 0.120,Y -484.518,Z 474.530,A 0.000,B 0.000,C 90.000,E1 95.334} C_DIS
LIN {X -0.201,Y -474.475,Z 474.523,A 0.000,B 0.000,C 90.000,E1 94.131} C_DIS
LIN {X -0.070,Y -457.007,Z 474.510,A 0.000,B 0.000,C 90.000,E1 91.835} C_DIS
LIN {X -0.137,Y -443.202,Z 474.499,A 0.000,B 0.000,C 90.000,E1 89.771} C_DIS
LIN {X 0.208,Y -431.666,Z 474.488,A 0.000,B 0.000,C 90.000,E1 87.879} C_DIS
LIN {X 0.119,Y -417.120,Z 474.475,A 0.000,B 0.000,C 90.000,E1 85.469} C_DIS
LIN {X 0.073,Y -404.503,Z 474.463,A 0.000,B 0.000,C 90.000,E1 83.280} C_DIS
LIN {X 0.111,Y -393.610,Z 474.452,A 0.000,B 0.000,C 90.000,E1 81.319} C_DIS
LIN {X 0.032,Y -382.716,Z 474.441,A 0.000,B 0.000,C 90.000,E1 79.342} C_DIS
LIN {X -0.115,Y -367.377,Z 474.425,A 0.000,B 0.000,C 90.000,E1 76.464} C_DIS
LIN {X -0.117,Y -357.303,Z 474.413,A 0.000,B 0.000,C 90.000,E1 74.393} C_DIS
LIN {X 0.119,Y -346.940,Z 474.400,A 0.000,B 0.000,C 90.000,E1 71.945} C_DIS
LIN {X -0.024,Y -335.310,Z 474.383,A 0.000,B 0.000,C 90.000,E1 68.901} C_DIS
LIN {X -0.133,Y -324.357,Z 474.365,A 0.000,B 0.000,C 90.000,E1 65.793} C_DIS
LIN {X -0.144,Y -315.781,Z 474.351,A 0.000,B 0.000,C 90.000,E1 63.256} C_DIS
LIN {X -0.086,Y -307.423,Z 474.337,A 0.000,B 0.000,C 90.000,E1 60.667} C_DIS
LIN {X -0.047,Y -299.218,Z 474.322,A 0.000,B 0.000,C 90.000,E1 58.043} C_DIS
LIN {X 0.102,Y -289.424,Z 474.304,A 0.000,B 0.000,C 90.000,E1 54.689} C_DIS
LIN {X 0.106,Y -282.026,Z 474.289,A 0.000,B 0.000,C 90.000,E1 51.984} C_DIS
LIN {X -0.168,Y -276.321,Z 474.278,A 0.000,B 0.000,C 90.000,E1 49.989} C_DIS
LIN {X 0.017,Y -270.265,Z 474.266,A 0.000,B 0.000,C 90.000,E1 47.877} C_DIS
LIN {X -0.130,Y -263.853,Z 474.254,A 0.000,B 0.000,C 90.000,E1 45.810} C_DIS
LIN {X -0.017,Y -257.233,Z 474.243,A 0.000,B 0.000,C 90.000,E1 43.662} C_DIS
LIN {X -0.017,Y -248.421,Z 474.227,A 0.000,B 0.000,C 90.000,E1 40.782} C_DIS
LIN {X -0.003,Y -237.758,Z 474.206,A 0.000,B 0.000,C 90.000,E1 37.111} C_DIS
LIN {X 0.012,Y -229.962,Z 474.190,A 0.000,B 0.000,C 90.000,E1 34.119} C_DIS
LIN {X 0.018,Y -222.962,Z 474.173,A 0.000,B 0.000,C 90.000,E1 31.082} C_DIS
LIN {X -0.070,Y -216.858,Z 474.156,A 0.000,B 0.000,C 90.000,E1 28.025} C_DIS
LIN {X -0.042,Y -211.502,Z 474.138,A 0.000,B 0.000,C 90.000,E1 24.899} C_DIS
LIN {X 0.078,Y -205.795,Z 474.116,A 0.000,B 0.000,C 90.000,E1 20.918} C_DIS
LIN {X 0.112,Y -201.147,Z 474.094,A 0.000,B 0.000,C 90.000,E1 16.913} C_DIS
LIN {X 0.096,Y -197.451,Z 474.072,A 0.000,B 0.000,C 90.000,E1 12.883} C_DIS
LIN {X -0.089,Y -193.997,Z 474.040,A 0.000,B 0.000,C 90.000,E1 7.239} C_DIS
LIN {X 0.103,Y -193.604,Z 473.961,A 0.000,B 0.000,C 90.000,E1 352.932} C_DIS
LIN {X 0.038,Y -197.018,Z 473.929,A 0.000,B 0.000,C 90.000,E1 347.229} C_DIS
LIN {X 0.043,Y -201.433,Z 473.902,A 0.000,B 0.000,C 90.000,E1 342.362} C_DIS
LIN {X -0.003,Y -206.088,Z 473.880,A 0.000,B 0.000,C 90.000,E1 338.358} C_DIS
LIN {X -0.097,Y -211.628,Z 473.858,A 0.000,B 0.000,C 90.000,E1 334.409} C_DIS
LIN {X -0.019,Y -217.843,Z 473.836,A 0.000,B 0.000,C 90.000,E1 330.461} C_DIS
LIN {X 0.009,Y -224.624,Z 473.814,A 0.000,B 0.000,C 90.000,E1 326.580} C_DIS
LIN {X 0.003,Y -232.152,Z 473.793,A 0.000,B 0.000,C 90.000,E1 322.763} C_DIS
LIN {X -0.031,Y -240.430,Z 473.772,A 0.000,B 0.000,C 90.000,E1 319.013} C_DIS
LIN {X 0.134,Y -248.865,Z 473.754,A 0.000,B 0.000,C 90.000,E1 315.648} C_DIS
LIN {X 0.042,Y -258.362,Z 473.736,A 0.000,B 0.000,C 90.000,E1 312.405} C_DIS
LIN {X 0.075,Y -268.936,Z 473.718,A 0.000,B 0.000,C 90.000,E1 309.197} C_DIS
LIN {X 0.042,Y -281.863,Z 473.699,A 0.000,B 0.000,C 90.000,E1 305.724} C_DIS
LIN {X -0.007,Y -295.798,Z 473.680,A 0.000,B 0.000,C 90.000,E1 302.339} C_DIS
LIN {X 0.097,Y -307.587,Z 473.665,A 0.000,B 0.000,C 90.000,E1 299.667} C_DIS
LIN {X 0.058,Y -320.301,Z 473.650,A 0.000,B 0.000,C 90.000,E1 297.078} C_DIS
LIN {X -0.150,Y -338.230,Z 473.633,A 0.000,B 0.000,C 90.000,E1 293.951} C_DIS
LIN {X -0.004,Y -352.145,Z 473.621,A 0.000,B 0.000,C 90.000,E1 291.770} C_DIS
LIN {X -0.188,Y -369.507,Z 473.608,A 0.000,B 0.000,C 90.000,E1 289.396} C_DIS
LIN {X 0.096,Y -390.838,Z 473.593,A 0.000,B 0.000,C 90.000,E1 286.732} C_DIS
LIN {X -0.177,Y -413.291,Z 473.579,A 0.000,B 0.000,C 90.000,E1 284.300} C_DIS
LIN {X 0.090,Y -428.412,Z 473.571,A 0.000,B 0.000,C 90.000,E1 282.715} C_DIS
LIN {X -0.165,Y -438.415,Z 473.565,A 0.000,B 0.000,C 90.000,E1 281.715} C_DIS
LIN {X -0.134,Y -448.057,Z 473.559,A 0.000,B 0.000,C 90.000,E1 280.658} C_DIS
LIN {X 0.068,Y -454.849,Z 473.555,A 0.000,B 0.000,C 90.000,E1 279.849} C_DIS
LIN {X 0.161,Y -463.075,Z 473.549,A 0.000,B 0.000,C 90.000,E1 278.803} C_DIS
LIN {X -0.116,Y -470.286,Z 473.543,A 0.000,B 0.000,C 90.000,E1 277.814} C_DIS
LIN {X -0.237,Y -475.026,Z 473.539,A 0.000,B 0.000,C 90.000,E1 277.068} C_DIS
LIN {X 0.225,Y -479.269,Z 473.535,A 0.000,B 0.000,C 90.000,E1 276.258} C_DIS
LIN {X 0.194,Y -482.944,Z 473.531,A 0.000,B 0.000,C 90.000,E1 275.511} C_DIS
LIN {X -0.114,Y -485.037,Z 473.528,A 0.000,B 0.000,C 90.000,E1 275.049} C_DIS
LIN {X 0.072,Y -486.818,Z 473.525,A 0.000,B 0.000,C 90.000,E1 274.531} C_DIS
LIN {X -0.224,Y -488.291,Z 473.522,A 0.000,B 0.000,C 90.000,E1 274.069} C_DIS
LIN {X -0.058,Y -489.467,Z 473.520,A 0.000,B 0.000,C 90.000,E1 273.555} C_DIS
LIN {X 0.148,Y -490.294,Z 473.517,A 0.000,B 0.000,C 90.000,E1 273.037} C_DIS
LIN {X -0.154,Y -490.768,Z 473.514,A 0.000,B 0.000,C 90.000,E1 272.579} C_DIS
LIN {X 0.041,Y -490.855,Z 473.512,A 0.000,B 0.000,C 90.000,E1 272.064} C_DIS
LIN {X -0.235,Y -490.521,Z 473.509,A 0.000,B 0.000,C 90.000,E1 271.604} C_DIS
LIN {X -0.036,Y -489.744,Z 473.506,A 0.000,B 0.000,C 90.000,E1 271.088} C_DIS
LIN {X 0.161,Y -488.471,Z 473.503,A 0.000,B 0.000,C 90.000,E1 270.573} C_DIS
LIN {X -0.133,Y -486.636,Z 473.501,A 0.000,B 0.000,C 90.000,E1 270.115} C_DIS
LIN {X 0.053,Y -484.118,Z 473.498,A 0.000,B 0.000,C 90.000,E1 269.599} C_DIS
LIN {X -0.105,Y -482.631,Z 473.496,A 0.000,B 0.000,C 90.000,E1 269.370} C_DIS
LIN {X 0.052,Y -478.970,Z 473.494,A 0.000,B 0.000,C 90.000,E1 268.854} C_DIS
LIN {X 0.189,Y -474.330,Z 473.491,A 0.000,B 0.000,C 90.000,E1 268.339} C_DIS
LIN {X -0.020,Y -468.803,Z 473.488,A 0.000,B 0.000,C 90.000,E1 267.879} C_DIS
LIN {X 0.167,Y -462.496,Z 473.486,A 0.000,B 0.000,C 90.000,E1 267.421} C_DIS
LIN {X -0.062,Y -455.969,Z 473.484,A 0.000,B 0.000,C 90.000,E1 267.078} C_DIS
LIN {X 0.162,Y -449.199,Z 473.482,A 0.000,B 0.000,C 90.000,E1 266.731} C_DIS
LIN {X -0.145,Y -442.073,Z 473.480,A 0.000,B 0.000,C 90.000,E1 266.502} C_DIS
LIN {X -0.069,Y -434.493,Z 473.479,A 0.000,B 0.000,C 90.000,E1 266.274} C_DIS
LIN {X -0.002,Y -425.639,Z 473.478,A 0.000,B 0.000,C 90.000,E1 266.102} C_DIS
LIN {X -0.147,Y -413.066,Z 473.478,A 0.000,B 0.000,C 90.000,E1 265.988} C_DIS
LIN {X 0.078,Y -405.558,Z 473.477,A 0.000,B 0.000,C 90.000,E1 265.927} C_DIS
LIN {X 0.013,Y -180.917,Z 473.477,A 0.000,B 0.000,C 90.000,E1 265.927} C_DIS
LIN {X -0.061,Y -180.872,Z 473.472,A 0.000,B 0.000,C 90.000,E1 265.065} C_DIS
LIN {X -0.004,Y -178.988,Z 473.444,A 0.000,B 0.000,C 90.000,E1 259.982} C_DIS
LIN {X 0.008,Y -177.969,Z 473.435,A 0.000,B 0.000,C 90.000,E1 258.285} C_DIS
LIN {X 0.027,Y -175.612,Z 473.411,A 0.000,B 0.000,C 90.000,E1 254.031} C_DIS
LIN {X 0.039,Y -172.334,Z 473.388,A 0.000,B 0.000,C 90.000,E1 249.752} C_DIS
LIN {X 0.017,Y -171.811,Z 473.383,A 0.000,B 0.000,C 90.000,E1 248.901} C_DIS
LIN {X 0.025,Y -170.274,Z 473.373,A 0.000,B 0.000,C 90.000,E1 247.177} C_DIS
LIN {X -0.039,Y -166.815,Z 473.349,A 0.000,B 0.000,C 90.000,E1 242.871} C_DIS
LIN {X 0.018,Y -162.797,Z 473.325,A 0.000,B 0.000,C 90.000,E1 238.486} C_DIS
LIN {X 0.079,Y -161.484,Z 473.315,A 0.000,B 0.000,C 90.000,E1 236.707} C_DIS
LIN {X -0.006,Y -157.480,Z 473.291,A 0.000,B 0.000,C 90.000,E1 232.316} C_DIS
LIN {X 0.051,Y -155.496,Z 473.276,A 0.000,B 0.000,C 90.000,E1 229.622} C_DIS
LIN {X -0.017,Y -151.802,Z 473.251,A 0.000,B 0.000,C 90.000,E1 225.162} C_DIS
LIN {X -0.005,Y -150.012,Z 473.236,A 0.000,B 0.000,C 90.000,E1 222.447} C_DIS
LIN {X 0.027,Y -146.837,Z 473.211,A 0.000,B 0.000,C 90.000,E1 217.890} C_DIS
LIN {X 0.013,Y -145.418,Z 473.195,A 0.000,B 0.000,C 90.000,E1 215.152} C_DIS
LIN {X 0.049,Y -142.846,Z 473.170,A 0.000,B 0.000,C 90.000,E1 210.541} C_DIS
LIN {X -0.021,Y -141.460,Z 473.149,A 0.000,B 0.000,C 90.000,E1 206.873} C_DIS
LIN {X 0.018,Y -139.374,Z 473.113,A 0.000,B 0.000,C 90.000,E1 200.355} C_DIS
LIN {X -0.040,Y -138.825,Z 473.098,A 0.000,B 0.000,C 90.000,E1 197.583} C_DIS
LIN {X 0.048,Y -138.353,Z 473.056,A 0.000,B 0.000,C 90.000,E1 190.074} C_DIS
LIN {X 0.022,Y -139.530,Z 473.004,A 0.000,B 0.000,C 90.000,E1 180.745} C_DIS
LIN {X -0.025,Y -141.210,Z 472.973,A 0.000,B 0.000,C 90.000,E1 175.179} C_DIS
LIN {X -0.067,Y -142.584,Z 472.958,A 0.000,B 0.000,C 90.000,E1 172.413} C_DIS
LIN {X 0.029,Y -144.880,Z 472.932,A 0.000,B 0.000,C 90.000,E1 167.757} C_DIS
LIN {X -0.017,Y -147.508,Z 472.912,A 0.000,B 0.000,C 90.000,E1 164.102} C_DIS
LIN {X 0.058,Y -150.099,Z 472.891,A 0.000,B 0.000,C 90.000,E1 160.423} C_DIS
LIN {X 0.070,Y -153.456,Z 472.871,A 0.000,B 0.000,C 90.000,E1 156.794} C_DIS
LIN {X -0.078,Y -157.819,Z 472.846,A 0.000,B 0.000,C 90.000,E1 152.359} C_DIS
LIN {X -0.047,Y -162.102,Z 472.827,A 0.000,B 0.000,C 90.000,E1 148.791} C_DIS
LIN {X -0.022,Y -166.302,Z 472.807,A 0.000,B 0.000,C 90.000,E1 145.261} C_DIS
LIN {X -0.025,Y -171.319,Z 472.788,A 0.000,B 0.000,C 90.000,E1 141.778} C_DIS
LIN {X 0.009,Y -176.219,Z 472.768,A 0.000,B 0.000,C 90.000,E1 138.324} C_DIS
LIN {X 0.003,Y -180.498,Z 472.754,A 0.000,B 0.000,C 90.000,E1 135.769} C_DIS
LIN {X -0.016,Y -185.900,Z 472.736,A 0.000,B 0.000,C 90.000,E1 132.405} C_DIS
LIN {X 0.045,Y -190.528,Z 472.722,A 0.000,B 0.000,C 90.000,E1 129.886} C_DIS
LIN {X 0.028,Y -193.922,Z 472.711,A 0.000,B 0.000,C 90.000,E1 127.890} C_DIS
LIN {X 0.006,Y -290.824,Z 472.711,A 0.000,B 0.000,C 90.000,E1 127.890} C_DIS
LIN {X 0.169,Y -293.825,Z 472.710,A 0.000,B 0.000,C 90.000,E1 127.810} C_DIS
LIN {X -0.077,Y -297.875,Z 472.709,A 0.000,B 0.000,C 90.000,E1 127.649} C_DIS
LIN {X -0.091,Y -300.264,Z 472.708,A 0.000,B 0.000,C 90.000,E1 127.443} C_DIS
LIN {X 0.006,Y -304.102,Z 472.705,A 0.000,B 0.000,C 90.000,E1 126.916} C_DIS
LIN {X 0.015,Y -305.841,Z 472.703,A 0.000,B 0.000,C 90.000,E1 126.583} C_DIS
LIN {X 0.025,Y -307.208,Z 472.701,A 0.000,B 0.000,C 90.000,E1 126.251} C_DIS
LIN {X 0.059,Y -318.563,Z 472.682,A 0.000,B 0.000,C 90.000,E1 122.673} C_DIS
LIN {X 0.127,Y -329.166,Z 472.666,A 0.000,B 0.000,C 90.000,E1 119.795} C_DIS
LIN {X 0.019,Y -341.139,Z 472.650,A 0.000,B 0.000,C 90.000,E1 117.001} C_DIS
LIN {X -0.067,Y -354.598,Z 472.635,A 0.000,B 0.000,C 90.000,E1 114.259} C_DIS
LIN {X 0.049,Y -367.903,Z 472.621,A 0.000,B 0.000,C 90.000,E1 111.844} C_DIS
LIN {X 0.023,Y -382.574,Z 472.608,A 0.000,B 0.000,C 90.000,E1 109.504} C_DIS
LIN {X -0.022,Y -398.714,Z 472.596,A 0.000,B 0.000,C 90.000,E1 107.221} C_DIS
LIN {X -0.169,Y -416.446,Z 472.583,A 0.000,B 0.000,C 90.000,E1 105.009} C_DIS
LIN {X -0.053,Y -435.841,Z 472.571,A 0.000,B 0.000,C 90.000,E1 102.827} C_DIS
LIN {X -0.231,Y -456.102,Z 472.560,A 0.000,B 0.000,C 90.000,E1 100.838} C_DIS
LIN {X -0.065,Y -476.894,Z 472.550,A 0.000,B 0.000,C 90.000,E1 98.973} C_DIS
LIN {X 0.142,Y -482.104,Z 472.547,A 0.000,B 0.000,C 90.000,E1 98.511} C_DIS
LIN {X -0.155,Y -485.735,Z 472.545,A 0.000,B 0.000,C 90.000,E1 98.106} C_DIS
LIN {X 0.207,Y -487.095,Z 472.544,A 0.000,B 0.000,C 90.000,E1 97.814} C_DIS
LIN {X 0.021,Y -488.102,Z 472.542,A 0.000,B 0.000,C 90.000,E1 97.587} C_DIS
LIN {X -0.258,Y -489.239,Z 472.539,A 0.000,B 0.000,C 90.000,E1 97.125} C_DIS
LIN {X -0.045,Y -489.365,Z 472.537,A 0.000,B 0.000,C 90.000,E1 96.606} C_DIS
LIN {X 0.176,Y -488.502,Z 472.534,A 0.000,B 0.000,C 90.000,E1 96.087} C_DIS
LIN {X -0.090,Y -486.498,Z 472.531,A 0.000,B 0.000,C 90.000,E1 95.625} C_DIS
LIN {X -0.202,Y -484.937,Z 472.530,A 0.000,B 0.000,C 90.000,E1 95.391} C_DIS
LIN {X -0.039,Y -474.929,Z 472.523,A 0.000,B 0.000,C 90.000,E1 94.131} C_DIS
LIN {X 0.096,Y -457.425,Z 472.510,A 0.000,B 0.000,C 90.000,E1 91.835} C_DIS
LIN {X -0.160,Y -445.212,Z 472.500,A 0.000,B 0.000,C 90.000,E1 90.057} C_DIS
LIN {X 0.209,Y -433.656,Z 472.490,A 0.000,B 0.000,C 90.000,E1 88.167} C_DIS
LIN {X -0.121,Y -417.473,Z 472.475,A 0.000,B 0.000,C 90.000,E1 85.527} C_DIS
LIN {X -0.151,Y -404.834,Z 472.463,A 0.000,B 0.000,C 90.000,E1 83.337} C_DIS
LIN {X -0.098,Y -393.958,Z 472.452,A 0.000,B 0.000,C 90.000,E1 81.376} C_DIS
LIN {X -0.122,Y -381.533,Z 472.439,A 0.000,B 0.000,C 90.000,E1 79.106} C_DIS
LIN {X 0.072,Y -367.753,Z 472.425,A 0.000,B 0.000,C 90.000,E1 76.464} C_DIS
LIN {X 0.024,Y -356.324,Z 472.412,A 0.000,B 0.000,C 90.000,E1 74.102} C_DIS
LIN {X 0.005,Y -346.055,Z 472.398,A 0.000,B 0.000,C 90.000,E1 71.692} C_DIS
LIN {X 0.162,Y -334.473,Z 472.381,A 0.000,B 0.000,C 90.000,E1 68.592} C_DIS
LIN {X 0.059,Y -324.558,Z 472.366,A 0.000,B 0.000,C 90.000,E1 65.793} C_DIS
LIN {X 0.047,Y -315.932,Z 472.351,A 0.000,B 0.000,C 90.000,E1 63.256} C_DIS
LIN {X 0.104,Y -307.543,Z 472.337,A 0.000,B 0.000,C 90.000,E1 60.667} C_DIS
LIN {X -0.017,Y -299.282,Z 472.323,A 0.000,B 0.000,C 90.000,E1 58.074} C_DIS
LIN {X -0.118,Y -289.457,Z 472.304,A 0.000,B 0.000,C 90.000,E1 54.769} C_DIS
LIN {X 0.063,Y -282.037,Z 472.289,A 0.000,B 0.000,C 90.000,E1 52.029} C_DIS
LIN {X 0.007,Y -276.329,Z 472.278,A 0.000,B 0.000,C 90.000,E1 49.989} C_DIS
LIN {X -0.011,Y -270.268,Z 472.266,A 0.000,B 0.000,C 90.000,E1 47.919} C_DIS
LIN {X 0.039,Y -263.894,Z 472.255,A 0.000,B 0.000,C 90.000,E1 45.810} C_DIS
LIN {X -0.038,Y -257.298,Z 472.243,A 0.000,B 0.000,C 90.000,E1 43.704} C_DIS
LIN {X -0.037,Y -250.690,Z 472.231,A 0.000,B 0.000,C 90.000,E1 41.553} C_DIS
LIN {X 0.035,Y -242.040,Z 472.215,A 0.000,B 0.000,C 90.000,E1 38.624} C_DIS
LIN {X -0.032,Y -233.870,Z 472.198,A 0.000,B 0.000,C 90.000,E1 35.678} C_DIS
LIN {X -0.060,Y -226.473,Z 472.181,A 0.000,B 0.000,C 90.000,E1 32.673} C_DIS
LIN {X -0.062,Y -219.879,Z 472.164,A 0.000,B 0.000,C 90.000,E1 29.617} C_DIS
LIN {X 0.005,Y -212.849,Z 472.143,A 0.000,B 0.000,C 90.000,E1 25.720} C_DIS
LIN {X 0.053,Y -206.898,Z 472.121,A 0.000,B 0.000,C 90.000,E1 21.770} C_DIS
LIN {X -0.073,Y -202.036,Z 472.099,A 0.000,B 0.000,C 90.000,E1 17.819} C_DIS
LIN {X -0.003,Y -198.104,Z 472.077,A 0.000,B 0.000,C 90.000,E1 13.772} C_DIS
LIN {X -0.067,Y -194.762,Z 472.049,A 0.000,B 0.000,C 90.000,E1 8.916} C_DIS
LIN {X -0.067,Y -192.263,Z 472.008,A 0.000,B 0.000,C 90.000,E1 1.547} C_DIS
LIN {X 0.040,Y -193.867,Z 471.956,A 0.000,B 0.000,C 90.000,E1 352.129} C_DIS
LIN {X 0.028,Y -196.868,Z 471.929,A 0.000,B 0.000,C 90.000,E1 347.229} C_DIS
LIN {X 0.025,Y -201.273,Z 471.902,A 0.000,B 0.000,C 90.000,E1 342.362} C_DIS
LIN {X 0.051,Y -205.924,Z 471.880,A 0.000,B 0.000,C 90.000,E1 338.337} C_DIS
LIN {X -0.124,Y -211.462,Z 471.858,A 0.000,B 0.000,C 90.000,E1 334.409} C_DIS
LIN {X -0.054,Y -217.690,Z 471.836,A 0.000,B 0.000,C 90.000,E1 330.461} C_DIS
LIN {X -0.031,Y -224.493,Z 471.814,A 0.000,B 0.000,C 90.000,E1 326.580} C_DIS
LIN {X -0.042,Y -232.020,Z 471.793,A 0.000,B 0.000,C 90.000,E1 322.763} C_DIS
LIN {X -0.082,Y -240.304,Z 471.772,A 0.000,B 0.000,C 90.000,E1 319.013} C_DIS
LIN {X 0.077,Y -248.748,Z 471.754,A 0.000,B 0.000,C 90.000,E1 315.648} C_DIS
LIN {X -0.021,Y -258.276,Z 471.736,A 0.000,B 0.000,C 90.000,E1 312.405} C_DIS
LIN {X 0.007,Y -268.869,Z 471.718,A 0.000,B 0.000,C 90.000,E1 309.197} C_DIS
LIN {X -0.030,Y -281.833,Z 471.698,A 0.000,B 0.000,C 90.000,E1 305.724} C_DIS
LIN {X -0.084,Y -295.791,Z 471.680,A 0.000,B 0.000,C 90.000,E1 302.339} C_DIS
LIN {X 0.048,Y -309.142,Z 471.663,A 0.000,B 0.000,C 90.000,E1 299.333} C_DIS
LIN {X -0.025,Y -320.337,Z 471.650,A 0.000,B 0.000,C 90.000,E1 297.078} C_DIS
LIN {X 0.072,Y -338.273,Z 471.633,A 0.000,B 0.000,C 90.000,E1 293.898} C_DIS
LIN {X -0.093,Y -352.201,Z 471.621,A 0.000,B 0.000,C 90.000,E1 291.770} C_DIS
LIN {X 0.191,Y -369.530,Z 471.608,A 0.000,B 0.000,C 90.000,E1 289.322} C_DIS
LIN {X 0.025,Y -393.393,Z 471.591,A 0.000,B 0.000,C 90.000,E1 286.441} C_DIS
LIN {X -0.237,Y -416.125,Z 471.578,A 0.000,B 0.000,C 90.000,E1 284.008} C_DIS
LIN {X -0.204,Y -431.131,Z 471.569,A 0.000,B 0.000,C 90.000,E1 282.479} C_DIS
LIN {X -0.051,Y -441.064,Z 471.563,A 0.000,B 0.000,C 90.000,E1 281.422} C_DIS
LIN {X 0.181,Y -448.250,Z 471.559,A 0.000,B 0.000,C 90.000,E1 280.602} C_DIS
LIN {X -0.059,Y -455.035,Z 471.555,A 0.000,B 0.000,C 90.000,E1 279.849} C_DIS
LIN {X 0.035,Y -463.254,Z 471.549,A 0.000,B 0.000,C 90.000,E1 278.803} C_DIS
LIN {X 0.225,Y -470.446,Z 471.543,A 0.000,B 0.000,C 90.000,E1 277.757} C_DIS
LIN {X 0.109,Y -475.196,Z 471.539,A 0.000,B 0.000,C 90.000,E1 277.011} C_DIS
LIN {X 0.100,Y -479.420,Z 471.535,A 0.000,B 0.000,C 90.000,E1 276.258} C_DIS
LIN {X 0.068,Y -483.087,Z 471.531,A 0.000,B 0.000,C 90.000,E1 275.511} C_DIS
LIN {X -0.239,Y -485.180,Z 471.528,A 0.000,B 0.000,C 90.000,E1 275.049} C_DIS
LIN {X -0.053,Y -486.983,Z 471.525,A 0.000,B 0.000,C 90.000,E1 274.531} C_DIS
LIN {X 0.138,Y -488.462,Z 471.522,A 0.000,B 0.000,C 90.000,E1 274.012} C_DIS
LIN {X -0.182,Y -489.635,Z 471.520,A 0.000,B 0.000,C 90.000,E1 273.555} C_DIS
LIN {X 0.025,Y -490.438,Z 471.517,A 0.000,B 0.000,C 90.000,E1 273.037} C_DIS
LIN {X 0.214,Y -490.904,Z 471.514,A 0.000,B 0.000,C 90.000,E1 272.522} C_DIS
LIN {X -0.080,Y -491.004,Z 471.511,A 0.000,B 0.000,C 90.000,E1 272.064} C_DIS
LIN {X 0.134,Y -490.652,Z 471.509,A 0.000,B 0.000,C 90.000,E1 271.547} C_DIS
LIN {X -0.156,Y -489.773,Z 471.506,A 0.000,B 0.000,C 90.000,E1 271.088} C_DIS
LIN {X 0.043,Y -488.551,Z 471.503,A 0.000,B 0.000,C 90.000,E1 270.573} C_DIS
LIN {X 0.235,Y -486.648,Z 471.500,A 0.000,B 0.000,C 90.000,E1 270.057} C_DIS
LIN {X -0.064,Y -484.153,Z 471.498,A 0.000,B 0.000,C 90.000,E1 269.599} C_DIS
LIN {X 0.103,Y -480.907,Z 471.495,A 0.000,B 0.000,C 90.000,E1 269.083} C_DIS
LIN {X -0.063,Y -478.970,Z 471.494,A 0.000,B 0.000,C 90.000,E1 268.854} C_DIS
LIN {X 0.074,Y -474.249,Z 471.491,A 0.000,B 0.000,C 90.000,E1 268.339} C_DIS
LIN {X -0.120,Y -468.676,Z 471.488,A 0.000,B 0.000,C 90.000,E1 267.879} C_DIS
LIN {X -0.155,Y -465.501,Z 471.487,A 0.000,B 0.000,C 90.000,E1 267.650} C_DIS
LIN {X -0.176,Y -458.959,Z 471.485,A 0.000,B 0.000,C 90.000,E1 267.249} C_DIS
LIN {X -0.149,Y -452.385,Z 471.483,A 0.000,B 0.000,C 90.000,E1 266.906} C_DIS
LIN {X 0.228,Y -445.213,Z 471.481,A 0.000,B 0.000,C 90.000,E1 266.560} C_DIS
LIN {X 0.113,Y -437.590,Z 471.480,A 0.000,B 0.000,C 90.000,E1 266.331} C_DIS
LIN {X 0.029,Y -429.750,Z 471.479,A 0.000,B 0.000,C 90.000,E1 266.159} C_DIS
LIN {X -0.100,Y -420.218,Z 471.478,A 0.000,B 0.000,C 90.000,E1 266.045} C_DIS
LIN {X -0.177,Y -412.497,Z 471.478,A 0.000,B 0.000,C 90.000,E1 265.988} C_DIS
LIN {X 0.099,Y -406.894,Z 471.477,A 0.000,B 0.000,C 90.000,E1 265.927} C_DIS
LIN {X 0.023,Y -180.917,Z 471.477,A 0.000,B 0.000,C 90.000,E1 265.927} C_DIS
LIN {X -0.066,Y -180.871,Z 471.472,A 0.000,B 0.000,C 90.000,E1 265.065} C_DIS
LIN {X -0.009,Y -178.988,Z 471.444,A 0.000,B 0.000,C 90.000,E1 259.982} C_DIS
LIN {X 0.002,Y -177.967,Z 471.435,A 0.000,B 0.000,C 90.000,E1 258.285} C_DIS
LIN {X 0.021,Y -175.611,Z 471.411,A 0.000,B 0.000,C 90.000,E1 254.031} C_DIS
LIN {X 0.033,Y -172.333,Z 471.388,A 0.000,B 0.000,C 90.000,E1 249.752} C_DIS
LIN {X 0.012,Y -171.810,Z 471.383,A 0.000,B 0.000,C 90.000,E1 248.901} C_DIS
LIN {X 0.019,Y -170.272,Z 471.373,A 0.000,B 0.000,C 90.000,E1 247.177} C_DIS
LIN {X -0.044,Y -166.813,Z 471.349,A 0.000,B 0.000,C 90.000,E1 242.871} C_DIS
LIN {X 0.012,Y -162.795,Z 471.325,A 0.000,B 0.000,C 90.000,E1 238.486} C_DIS
LIN {X 0.073,Y -161.483,Z 471.315,A 0.000,B 0.000,C 90.000,E1 236.707} C_DIS
LIN {X -0.011,Y -157.478,Z 471.291,A 0.000,B 0.000,C 90.000,E1 232.316} C_DIS
LIN {X 0.046,Y -155.495,Z 471.276,A 0.000,B 0.000,C 90.000,E1 229.622} C_DIS
LIN {X -0.022,Y -151.801,Z 471.251,A 0.000,B 0.000,C 90.000,E1 225.162} C_DIS
LIN {X -0.010,Y -150.010,Z 471.236,A 0.000,B 0.000,C 90.000,E1 222.447} C_DIS
LIN {X 0.022,Y -146.836,Z 471.211,A 0.000,B 0.000,C 90.000,E1 217.890} C_DIS
LIN {X 0.008,Y -145.417,Z 471.195,A 0.000,B 0.000,C 90.000,E1 215.152} C_DIS
LIN {X 0.044,Y -142.845,Z 471.170,A 0.000,B 0.000,C 90.000,E1 210.541} C_DIS
LIN {X -0.027,Y -141.460,Z 471.149,A 0.000,B 0.000,C 90.000,E1 206.873} C_DIS
LIN {X 0.013,Y -139.375,Z 471.113,A 0.000,B 0.000,C 90.000,E1 200.355} C_DIS
LIN {X -0.044,Y -138.824,Z 471.098,A 0.000,B 0.000,C 90.000,E1 197.583} C_DIS
LIN {X 0.044,Y -138.353,Z 471.056,A 0.000,B 0.000,C 90.000,E1 190.074} C_DIS
LIN {X 0.017,Y -139.531,Z 471.004,A 0.000,B 0.000,C 90.000,E1 180.745} C_DIS
LIN {X -0.030,Y -141.210,Z 470.973,A 0.000,B 0.000,C 90.000,E1 175.179} C_DIS
LIN {X 0.070,Y -142.585,Z 470.958,A 0.000,B 0.000,C 90.000,E1 172.356} C_DIS
LIN {X 0.025,Y -144.882,Z 470.932,A 0.000,B 0.000,C 90.000,E1 167.757} C_DIS
LIN {X -0.022,Y -147.508,Z 470.912,A 0.000,B 0.000,C 90.000,E1 164.102} C_DIS
LIN {X 0.052,Y -150.101,Z 470.891,A 0.000,B 0.000,C 90.000,E1 160.423} C_DIS
LIN {X 0.065,Y -153.458,Z 470.871,A 0.000,B 0.000,C 90.000,E1 156.794} C_DIS
LIN {X -0.083,Y -157.821,Z 470.846,A 0.000,B 0.000,C 90.000,E1 152.359} C_DIS
LIN {X -0.052,Y -162.105,Z 470.827,A 0.000,B 0.000,C 90.000,E1 148.791} C_DIS
LIN {X -0.028,Y -166.305,Z 470.807,A 0.000,B 0.000,C 90.000,E1 145.261} C_DIS
LIN {X -0.031,Y -171.322,Z 470.788,A 0.000,B 0.000,C 90.000,E1 141.778} C_DIS
LIN {X 0.004,Y -176.222,Z 470.768,A 0.000,B 0.000,C 90.000,E1 138.324} C_DIS
LIN {X -0.003,Y -180.500,Z 470.754,A 0.000,B 0.000,C 90.000,E1 135.769} C_DIS
LIN {X -0.022,Y -185.904,Z 470.736,A 0.000,B 0.000,C 90.000,E1 132.405} C_DIS
LIN {X 0.039,Y -190.531,Z 470.722,A 0.000,B 0.000,C 90.000,E1 129.886} C_DIS
LIN {X -0.021,Y -194.009,Z 470.710,A 0.000,B 0.000,C 90.000,E1 127.855} C_DIS
LIN {X 0.155,Y -291.263,Z 470.710,A 0.000,B 0.000,C 90.000,E1 127.810} C_DIS
LIN {X -0.088,Y -297.313,Z 470.709,A 0.000,B 0.000,C 90.000,E1 127.649} C_DIS
LIN {X -0.101,Y -299.906,Z 470.708,A 0.000,B 0.000,C 90.000,E1 127.443} C_DIS
LIN {X -0.003,Y -303.719,Z 470.705,A 0.000,B 0.000,C 90.000,E1 126.950} C_DIS
LIN {X 0.188,Y -305.573,Z 470.703,A 0.000,B 0.000,C 90.000,E1 126.583} C_DIS
LIN {X -0.050,Y -307.024,Z 470.702,A 0.000,B 0.000,C 90.000,E1 126.297} C_DIS
LIN {X -0.062,Y -309.123,Z 470.698,A 0.000,B 0.000,C 90.000,E1 125.644} C_DIS
LIN {X -0.137,Y -319.547,Z 470.680,A 0.000,B 0.000,C 90.000,E1 122.418} C_DIS
LIN {X -0.037,Y -330.281,Z 470.664,A 0.000,B 0.000,C 90.000,E1 119.539} C_DIS
LIN {X -0.121,Y -342.401,Z 470.648,A 0.000,B 0.000,C 90.000,E1 116.744} C_DIS
LIN {X 0.153,Y -356.011,Z 470.633,A 0.000,B 0.000,C 90.000,E1 113.951} C_DIS
LIN {X -0.028,Y -369.464,Z 470.620,A 0.000,B 0.000,C 90.000,E1 111.589} C_DIS
LIN {X -0.151,Y -384.293,Z 470.607,A 0.000,B 0.000,C 90.000,E1 109.268} C_DIS
LIN {X -0.153,Y -400.608,Z 470.594,A 0.000,B 0.000,C 90.000,E1 106.985} C_DIS
LIN {X 0.148,Y -418.527,Z 470.582,A 0.000,B 0.000,C 90.000,E1 104.717} C_DIS
LIN {X -0.045,Y -438.061,Z 470.570,A 0.000,B 0.000,C 90.000,E1 102.591} C_DIS
LIN {X -0.069,Y -458.386,Z 470.559,A 0.000,B 0.000,C 90.000,E1 100.602} C_DIS
LIN {X -0.163,Y -481.866,Z 470.547,A 0.000,B 0.000,C 90.000,E1 98.568} C_DIS
LIN {X -0.090,Y -484.006,Z 470.546,A 0.000,B 0.000,C 90.000,E1 98.341} C_DIS
LIN {X 0.055,Y -485.641,Z 470.545,A 0.000,B 0.000,C 90.000,E1 98.106} C_DIS
LIN {X -0.060,Y -487.066,Z 470.544,A 0.000,B 0.000,C 90.000,E1 97.871} C_DIS
LIN {X -0.242,Y -488.126,Z 470.542,A 0.000,B 0.000,C 90.000,E1 97.644} C_DIS
LIN {X -0.037,Y -489.358,Z 470.540,A 0.000,B 0.000,C 90.000,E1 97.125} C_DIS
LIN {X 0.177,Y -489.571,Z 470.537,A 0.000,B 0.000,C 90.000,E1 96.606} C_DIS
LIN {X -0.088,Y -488.795,Z 470.534,A 0.000,B 0.000,C 90.000,E1 96.144} C_DIS
LIN {X 0.133,Y -486.901,Z 470.531,A 0.000,B 0.000,C 90.000,E1 95.625} C_DIS
LIN {X 0.020,Y -485.415,Z 470.530,A 0.000,B 0.000,C 90.000,E1 95.391} C_DIS
LIN {X -0.119,Y -477.469,Z 470.524,A 0.000,B 0.000,C 90.000,E1 94.416} C_DIS
LIN {X 0.083,Y -459.771,Z 470.512,A 0.000,B 0.000,C 90.000,E1 92.121} C_DIS
LIN {X -0.135,Y -447.296,Z 470.502,A 0.000,B 0.000,C 90.000,E1 90.344} C_DIS
LIN {X 0.009,Y -434.047,Z 470.490,A 0.000,B 0.000,C 90.000,E1 88.224} C_DIS
LIN {X 0.115,Y -417.859,Z 470.475,A 0.000,B 0.000,C 90.000,E1 85.527} C_DIS
LIN {X 0.140,Y -403.670,Z 470.462,A 0.000,B 0.000,C 90.000,E1 83.053} C_DIS
LIN {X -0.180,Y -392.778,Z 470.451,A 0.000,B 0.000,C 90.000,E1 81.141} C_DIS
LIN {X 0.119,Y -381.940,Z 470.440,A 0.000,B 0.000,C 90.000,E1 79.106} C_DIS
LIN {X -0.042,Y -368.180,Z 470.425,A 0.000,B 0.000,C 90.000,E1 76.520} C_DIS
LIN {X -0.073,Y -356.739,Z 470.412,A 0.000,B 0.000,C 90.000,E1 74.157} C_DIS
LIN {X -0.160,Y -345.205,Z 470.397,A 0.000,B 0.000,C 90.000,E1 71.456} C_DIS
LIN {X 0.092,Y -333.662,Z 470.380,A 0.000,B 0.000,C 90.000,E1 68.337} C_DIS
LIN {X -0.030,Y -323.713,Z 470.364,A 0.000,B 0.000,C 90.000,E1 65.537} C_DIS
LIN {X -0.003,Y -316.124,Z 470.352,A 0.000,B 0.000,C 90.000,E1 63.307} C_DIS
LIN {X 0.065,Y -307.688,Z 470.337,A 0.000,B 0.000,C 90.000,E1 60.717} C_DIS
LIN {X -0.045,Y -299.379,Z 470.323,A 0.000,B 0.000,C 90.000,E1 58.122} C_DIS
LIN {X 0.104,Y -289.515,Z 470.304,A 0.000,B 0.000,C 90.000,E1 54.769} C_DIS
LIN {X -0.115,Y -282.082,Z 470.289,A 0.000,B 0.000,C 90.000,E1 52.110} C_DIS
LIN {X 0.010,Y -276.366,Z 470.278,A 0.000,B 0.000,C 90.000,E1 50.033} C_DIS
LIN {X 0.018,Y -270.303,Z 470.266,A 0.000,B 0.000,C 90.000,E1 47.957} C_DIS
LIN {X -0.129,Y -263.946,Z 470.255,A 0.000,B 0.000,C 90.000,E1 45.891} C_DIS
LIN {X 0.158,Y -257.374,Z 470.243,A 0.000,B 0.000,C 90.000,E1 43.704} C_DIS
LIN {X -0.046,Y -250.792,Z 470.231,A 0.000,B 0.000,C 90.000,E1 41.595} C_DIS
LIN {X 0.020,Y -242.142,Z 470.215,A 0.000,B 0.000,C 90.000,E1 38.669} C_DIS
LIN {X -0.051,Y -233.981,Z 470.198,A 0.000,B 0.000,C 90.000,E1 35.724} C_DIS
LIN {X 0.109,Y -226.581,Z 470.182,A 0.000,B 0.000,C 90.000,E1 32.673} C_DIS
LIN {X -0.087,Y -219.966,Z 470.165,A 0.000,B 0.000,C 90.000,E1 29.667} C_DIS
LIN {X 0.022,Y -214.238,Z 470.147,A 0.000,B 0.000,C 90.000,E1 26.539} C_DIS
LIN {X -0.080,Y -208.064,Z 470.126,A 0.000,B 0.000,C 90.000,E1 22.642} C_DIS
LIN {X -0.030,Y -202.941,Z 470.104,A 0.000,B 0.000,C 90.000,E1 18.652} C_DIS
LIN {X 0.113,Y -198.811,Z 470.081,A 0.000,B 0.000,C 90.000,E1 14.592} C_DIS
LIN {X 0.103,Y -195.183,Z 470.054,A 0.000,B 0.000,C 90.000,E1 9.726} C_DIS
LIN {X 0.003,Y -192.458,Z 470.018,A 0.000,B 0.000,C 90.000,E1 3.212} C_DIS
LIN {X 0.034,Y -193.742,Z 469.956,A 0.000,B 0.000,C 90.000,E1 352.129} C_DIS
LIN {X 0.016,Y -196.735,Z 469.929,A 0.000,B 0.000,C 90.000,E1 347.229} C_DIS
LIN {X 0.008,Y -201.117,Z 469.902,A 0.000,B 0.000,C 90.000,E1 342.362} C_DIS
LIN {X 0.029,Y -205.761,Z 469.880,A 0.000,B 0.000,C 90.000,E1 338.337} C_DIS
LIN {X 0.038,Y -211.283,Z 469.858,A 0.000,B 0.000,C 90.000,E1 334.357} C_DIS
LIN {X -0.088,Y -217.534,Z 469.836,A 0.000,B 0.000,C 90.000,E1 330.461} C_DIS
LIN {X 0.023,Y -222.964,Z 469.819,A 0.000,B 0.000,C 90.000,E1 327.327} C_DIS
LIN {X 0.017,Y -230.299,Z 469.797,A 0.000,B 0.000,C 90.000,E1 323.497} C_DIS
LIN {X -0.077,Y -238.430,Z 469.776,A 0.000,B 0.000,C 90.000,E1 319.747} C_DIS
LIN {X 0.055,Y -245.706,Z 469.760,A 0.000,B 0.000,C 90.000,E1 316.743} C_DIS
LIN {X 0.028,Y -254.867,Z 469.741,A 0.000,B 0.000,C 90.000,E1 313.461} C_DIS
LIN {X -0.051,Y -265.169,Z 469.724,A 0.000,B 0.000,C 90.000,E1 310.253} C_DIS
LIN {X 0.037,Y -276.466,Z 469.706,A 0.000,B 0.000,C 90.000,E1 307.076} C_DIS
LIN {X 0.004,Y -288.666,Z 469.689,A 0.000,B 0.000,C 90.000,E1 303.992} C_DIS
